    movel([0.074440, -1.320583, -2.610571, -0.781234, 1.570796, 1.645237],accel_mss,speed_ms,0,blend_radius_m)
    movel([0.074315, -1.320855, -2.610402, -0.781132, 1.570796, 1.645112],accel_mss,speed_ms,0,blend_radius_m)
    movel([0.073757, -1.321736, -2.609852, -0.780801, 1.570796, 1.644553],accel_mss,speed_ms,0,blend_radius_m)
    movel([0.073104, -1.322417, -2.609427, -0.780545, 1.570796, 1.643900],accel_mss,speed_ms,0,blend_radius_m)
    movel([0.072314, -1.322927, -2.609108, -0.780355, 1.570796, 1.643111],accel_mss,speed_ms,0,blend_radius_m)
    movel([0.071362, -1.323294, -2.608878, -0.780217, 1.570796, 1.642159],accel_mss,speed_ms,0,blend_radius_m)
    movel([0.070869, -1.323423, -2.608797, -0.780169, 1.570796, 1.641665],accel_mss,speed_ms,0,blend_radius_m)
    movel([0.070526, -1.323474, -2.608765, -0.780150, 1.570796, 1.641322],accel_mss,speed_ms,0,blend_radius_m)
    movel([0.070234, -1.323465, -2.608771, -0.780154, 1.570796, 1.641030],accel_mss,speed_ms,0,blend_radius_m)
    movel([0.069916, -1.323397, -2.608813, -0.780179, 1.570796, 1.640712],accel_mss,speed_ms,0,blend_radius_m)
    movel([0.069099, -1.322793, -2.609191, -0.780404, 1.570796, 1.639896],accel_mss,speed_ms,0,blend_radius_m)
    movel([0.068874, -1.321709, -2.609869, -0.780811, 1.570796, 1.639671],accel_mss,speed_ms,0,blend_radius_m)
    movel([0.069290, -1.320407, -2.610681, -0.781301, 1.570796, 1.640086],accel_mss,speed_ms,0,blend_radius_m)
    movel([0.070255, -1.319201, -2.611431, -0.781757, 1.570796, 1.641051],accel_mss,speed_ms,0,blend_radius_m)
    movel([0.070604, -1.318907, -2.611613, -0.781868, 1.570796, 1.641400],accel_mss,speed_ms,0,blend_radius_m)
    movel([0.070915, -1.318695, -2.611745, -0.781949, 1.570796, 1.641711],accel_mss,speed_ms,0,blend_radius_m)
    movel([0.071271, -1.318512, -2.611859, -0.782018, 1.570796, 1.642068],accel_mss,speed_ms,0,blend_radius_m)
    movel([0.071774, -1.318306, -2.611986, -0.782096, 1.570796, 1.642570],accel_mss,speed_ms,0,blend_radius_m)
    movel([0.072472, -1.318085, -2.612123, -0.782180, 1.570796, 1.643268],accel_mss,speed_ms,0,blend_radius_m)
    movel([0.073056, -1.318004, -2.612174, -0.782212, 1.570796, 1.643852],accel_mss,speed_ms,0,blend_radius_m)
    movel([0.073553, -1.318057, -2.612141, -0.782191, 1.570796, 1.644349],accel_mss,speed_ms,0,blend_radius_m)
    movel([0.073982, -1.318249, -2.612022, -0.782118, 1.570796, 1.644779],accel_mss,speed_ms,0,blend_radius_m)
    movel([0.074267, -1.318512, -2.611859, -0.782018, 1.570796, 1.645063],accel_mss,speed_ms,0,blend_radius_m)
    movel([0.074500, -1.318909, -2.611612, -0.781868, 1.570796, 1.645296],accel_mss,speed_ms,0,blend_radius_m)
    movel([0.074648, -1.319355, -2.611336, -0.781699, 1.570796, 1.645444],accel_mss,speed_ms,0,blend_radius_m)
    speed_ms = 0.003
    movel([0.074648, -1.322804, -2.612923, -0.776662, 1.570796, 1.645444],accel_mss,speed_ms,0,blend_radius_m)
    speed_ms = 0.007
    movel([0.074675, -1.323216, -2.612666, -0.776507, 1.570796, 1.645472],accel_mss,speed_ms,0,blend_radius_m)
    movel([0.074553, -1.323727, -2.612346, -0.776316, 1.570796, 1.645349],accel_mss,speed_ms,0,blend_radius_m)
    movel([0.074440, -1.324030, -2.612157, -0.776203, 1.570796, 1.645237],accel_mss,speed_ms,0,blend_radius_m)
    movel([0.074315, -1.324301, -2.611987, -0.776101, 1.570796, 1.645112],accel_mss,speed_ms,0,blend_radius_m)
    movel([0.073757, -1.325180, -2.611436, -0.775773, 1.570796, 1.644553],accel_mss,speed_ms,0,blend_radius_m)
    movel([0.073104, -1.325859, -2.611009, -0.775521, 1.570796, 1.643900],accel_mss,speed_ms,0,blend_radius_m)
    movel([0.072314, -1.326368, -2.610689, -0.775332, 1.570796, 1.643111],accel_mss,speed_ms,0,blend_radius_m)
    movel([0.071362, -1.326734, -2.610459, -0.775196, 1.570796, 1.642159],accel_mss,speed_ms,0,blend_radius_m)
    movel([0.070869, -1.326862, -2.610378, -0.775149, 1.570796, 1.641665],accel_mss,speed_ms,0,blend_radius_m)
    movel([0.070526, -1.326913, -2.610346, -0.775130, 1.570796, 1.641322],accel_mss,speed_ms,0,blend_radius_m)
    movel([0.070234, -1.326904, -2.610351, -0.775133, 1.570796, 1.641030],accel_mss,speed_ms,0,blend_radius_m)
    movel([0.069916, -1.326837, -2.610394, -0.775159, 1.570796, 1.640712],accel_mss,speed_ms,0,blend_radius_m)
    movel([0.069099, -1.326234, -2.610773, -0.775382, 1.570796, 1.639896],accel_mss,speed_ms,0,blend_radius_m)
    movel([0.068874, -1.325153, -2.611453, -0.775784, 1.570796, 1.639671],accel_mss,speed_ms,0,blend_radius_m)
    movel([0.069290, -1.323854, -2.612267, -0.776268, 1.570796, 1.640086],accel_mss,speed_ms,0,blend_radius_m)
    movel([0.070255, -1.322650, -2.613019, -0.776720, 1.570796, 1.641051],accel_mss,speed_ms,0,blend_radius_m)
    movel([0.070604, -1.322358, -2.613202, -0.776829, 1.570796, 1.641400],accel_mss,speed_ms,0,blend_radius_m)
    movel([0.070915, -1.322146, -2.613334, -0.776909, 1.570796, 1.641711],accel_mss,speed_ms,0,blend_radius_m)
    movel([0.071271, -1.321963, -2.613448, -0.776978, 1.570796, 1.642068],accel_mss,speed_ms,0,blend_radius_m)
    movel([0.071774, -1.321758, -2.613576, -0.777055, 1.570796, 1.642570],accel_mss,speed_ms,0,blend_radius_m)
    movel([0.072472, -1.321538, -2.613713, -0.777138, 1.570796, 1.643268],accel_mss,speed_ms,0,blend_radius_m)
    movel([0.073056, -1.321456, -2.613764, -0.777169, 1.570796, 1.643852],accel_mss,speed_ms,0,blend_radius_m)
    movel([0.073553, -1.321509, -2.613731, -0.777149, 1.570796, 1.644349],accel_mss,speed_ms,0,blend_radius_m)
    movel([0.073982, -1.321701, -2.613611, -0.777077, 1.570796, 1.644779],accel_mss,speed_ms,0,blend_radius_m)
    movel([0.074267, -1.321963, -2.613448, -0.776978, 1.570796, 1.645063],accel_mss,speed_ms,0,blend_radius_m)
    movel([0.074500, -1.322359, -2.613201, -0.776829, 1.570796, 1.645296],accel_mss,speed_ms,0,blend_radius_m)
    movel([0.074648, -1.322804, -2.612923, -0.776662, 1.570796, 1.645444],accel_mss,speed_ms,0,blend_radius_m)
    speed_ms = 0.003
    movel([0.074648, -1.309165, -2.606523, -0.796701, 1.570796, 1.645444],accel_mss,speed_ms,0,blend_radius_m)
    speed_ms = 1.000
    movel([0.074648, -1.283142, -2.593332, -0.835915, 1.570796, 1.645444],accel_mss,speed_ms,0,blend_radius_m)
    movel([0.075024, -1.282687, -2.593600, -0.836102, 1.570796, 1.645820],accel_mss,speed_ms,0,blend_radius_m)
    movel([0.075024, -1.308718, -2.606796, -0.796875, 1.570796, 1.645820],accel_mss,speed_ms,0,blend_radius_m)
    speed_ms = 0.003
    movel([0.075024, -1.318910, -2.611612, -0.781867, 1.570796, 1.645820],accel_mss,speed_ms,0,blend_radius_m)
    speed_ms = 0.007
    movel([0.075085, -1.319510, -2.611239, -0.781640, 1.570796, 1.645881],accel_mss,speed_ms,0,blend_radius_m)
    movel([0.074948, -1.320246, -2.610781, -0.781362, 1.570796, 1.645744],accel_mss,speed_ms,0,blend_radius_m)
    movel([0.074641, -1.321022, -2.610298, -0.781069, 1.570796, 1.645437],accel_mss,speed_ms,0,blend_radius_m)
    movel([0.074198, -1.321742, -2.609848, -0.780798, 1.570796, 1.644994],accel_mss,speed_ms,0,blend_radius_m)
    movel([0.073687, -1.322309, -2.609494, -0.780586, 1.570796, 1.644483],accel_mss,speed_ms,0,blend_radius_m)
    movel([0.073025, -1.322849, -2.609156, -0.780384, 1.570796, 1.643822],accel_mss,speed_ms,0,blend_radius_m)
    movel([0.072291, -1.323304, -2.608871, -0.780213, 1.570796, 1.643087],accel_mss,speed_ms,0,blend_radius_m)
    movel([0.071565, -1.323618, -2.608674, -0.780096, 1.570796, 1.642362],accel_mss,speed_ms,0,blend_radius_m)
    movel([0.070602, -1.323847, -2.608531, -0.780011, 1.570796, 1.641398],accel_mss,speed_ms,0,blend_radius_m)
    movel([0.069813, -1.323830, -2.608542, -0.780017, 1.570796, 1.640609],accel_mss,speed_ms,0,blend_radius_m)
    movel([0.069187, -1.323555, -2.608714, -0.780120, 1.570796, 1.639984],accel_mss,speed_ms,0,blend_radius_m)
    movel([0.068697, -1.323026, -2.609045, -0.780317, 1.570796, 1.639493],accel_mss,speed_ms,0,blend_radius_m)
    movel([0.068546, -1.322743, -2.609223, -0.780423, 1.570796, 1.639343],accel_mss,speed_ms,0,blend_radius_m)
    movel([0.068478, -1.322487, -2.609383, -0.780519, 1.570796, 1.639274],accel_mss,speed_ms,0,blend_radius_m)
    movel([0.068472, -1.322167, -2.609583, -0.780639, 1.570796, 1.639268],accel_mss,speed_ms,0,blend_radius_m)
    movel([0.068526, -1.321647, -2.609908, -0.780834, 1.570796, 1.639322],accel_mss,speed_ms,0,blend_radius_m)
    movel([0.068607, -1.321120, -2.610237, -0.781032, 1.570796, 1.639403],accel_mss,speed_ms,0,blend_radius_m)
    movel([0.068702, -1.320774, -2.610453, -0.781163, 1.570796, 1.639499],accel_mss,speed_ms,0,blend_radius_m)
    movel([0.068847, -1.320465, -2.610645, -0.781279, 1.570796, 1.639644],accel_mss,speed_ms,0,blend_radius_m)
    movel([0.069093, -1.320085, -2.610882, -0.781423, 1.570796, 1.639889],accel_mss,speed_ms,0,blend_radius_m)
    movel([0.069307, -1.319800, -2.611058, -0.781530, 1.570796, 1.640103],accel_mss,speed_ms,0,blend_radius_m)
    movel([0.069588, -1.319471, -2.611263, -0.781655, 1.570796, 1.640384],accel_mss,speed_ms,0,blend_radius_m)
    movel([0.069884, -1.319150, -2.611463, -0.781776, 1.570796, 1.640680],accel_mss,speed_ms,0,blend_radius_m)
    movel([0.070148, -1.318894, -2.611621, -0.781873, 1.570796, 1.640945],accel_mss,speed_ms,0,blend_radius_m)
    movel([0.070517, -1.318583, -2.611815, -0.781991, 1.570796, 1.641314],accel_mss,speed_ms,0,blend_radius_m)
    movel([0.070837, -1.318370, -2.611946, -0.782072, 1.570796, 1.641633],accel_mss,speed_ms,0,blend_radius_m)
    movel([0.071214, -1.318184, -2.612062, -0.782143, 1.570796, 1.642011],accel_mss,speed_ms,0,blend_radius_m)
    movel([0.071809, -1.317950, -2.612207, -0.782232, 1.570796, 1.642605],accel_mss,speed_ms,0,blend_radius_m)
    movel([0.072379, -1.317746, -2.612333, -0.782309, 1.570796, 1.643176],accel_mss,speed_ms,0,blend_radius_m)
    movel([0.072764, -1.317643, -2.612397, -0.782349, 1.570796, 1.643560],accel_mss,speed_ms,0,blend_radius_m)
    movel([0.073074, -1.317602, -2.612422, -0.782364, 1.570796, 1.643870],accel_mss,speed_ms,0,blend_radius_m)
    movel([0.073396, -1.317616, -2.612414, -0.782359, 1.570796, 1.644192],accel_mss,speed_ms,0,blend_radius_m)
    movel([0.073967, -1.317754, -2.612329, -0.782307, 1.570796, 1.644763],accel_mss,speed_ms,0,blend_radius_m)
    movel([0.074437, -1.318021, -2.612163, -0.782205, 1.570796, 1.645234],accel_mss,speed_ms,0,blend_radius_m)
    movel([0.074794, -1.318414, -2.611920, -0.782056, 1.570796, 1.645591],accel_mss,speed_ms,0,blend_radius_m)
    movel([0.075024, -1.318910, -2.611612, -0.781867, 1.570796, 1.645820],accel_mss,speed_ms,0,blend_radius_m)
    speed_ms = 0.003
    movel([0.075024, -1.322360, -2.613200, -0.776828, 1.570796, 1.645820],accel_mss,speed_ms,0,blend_radius_m)
    speed_ms = 0.007
    movel([0.075085, -1.322959, -2.612826, -0.776604, 1.570796, 1.645881],accel_mss,speed_ms,0,blend_radius_m)
    movel([0.074948, -1.323693, -2.612367, -0.776328, 1.570796, 1.645744],accel_mss,speed_ms,0,blend_radius_m)
    movel([0.074641, -1.324467, -2.611883, -0.776039, 1.570796, 1.645437],accel_mss,speed_ms,0,blend_radius_m)
    movel([0.074198, -1.325186, -2.611432, -0.775771, 1.570796, 1.644994],accel_mss,speed_ms,0,blend_radius_m)
    movel([0.073687, -1.325751, -2.611077, -0.775561, 1.570796, 1.644483],accel_mss,speed_ms,0,blend_radius_m)
    movel([0.073025, -1.326290, -2.610738, -0.775361, 1.570796, 1.643822],accel_mss,speed_ms,0,blend_radius_m)
    movel([0.072291, -1.326744, -2.610452, -0.775193, 1.570796, 1.643087],accel_mss,speed_ms,0,blend_radius_m)
    movel([0.071565, -1.327058, -2.610255, -0.775077, 1.570796, 1.642362],accel_mss,speed_ms,0,blend_radius_m)
    movel([0.070602, -1.327285, -2.610111, -0.774992, 1.570796, 1.641398],accel_mss,speed_ms,0,blend_radius_m)
    movel([0.069813, -1.327269, -2.610122, -0.774999, 1.570796, 1.640609],accel_mss,speed_ms,0,blend_radius_m)
    movel([0.069187, -1.326994, -2.610295, -0.775100, 1.570796, 1.639984],accel_mss,speed_ms,0,blend_radius_m)
    movel([0.068697, -1.326467, -2.610627, -0.775296, 1.570796, 1.639493],accel_mss,speed_ms,0,blend_radius_m)
    movel([0.068546, -1.326184, -2.610804, -0.775400, 1.570796, 1.639343],accel_mss,speed_ms,0,blend_radius_m)
    movel([0.068478, -1.325929, -2.610965, -0.775495, 1.570796, 1.639274],accel_mss,speed_ms,0,blend_radius_m)
    movel([0.068472, -1.325610, -2.611166, -0.775614, 1.570796, 1.639268],accel_mss,speed_ms,0,blend_radius_m)
    movel([0.068526, -1.325091, -2.611492, -0.775807, 1.570796, 1.639322],accel_mss,speed_ms,0,blend_radius_m)
    movel([0.068607, -1.324565, -2.611821, -0.776003, 1.570796, 1.639403],accel_mss,speed_ms,0,blend_radius_m)
    movel([0.068702, -1.324220, -2.612038, -0.776132, 1.570796, 1.639499],accel_mss,speed_ms,0,blend_radius_m)
    movel([0.068847, -1.323912, -2.612230, -0.776247, 1.570796, 1.639644],accel_mss,speed_ms,0,blend_radius_m)
    movel([0.069093, -1.323532, -2.612468, -0.776389, 1.570796, 1.639889],accel_mss,speed_ms,0,blend_radius_m)
    movel([0.069307, -1.323249, -2.612645, -0.776495, 1.570796, 1.640103],accel_mss,speed_ms,0,blend_radius_m)
    movel([0.069588, -1.322920, -2.612851, -0.776618, 1.570796, 1.640384],accel_mss,speed_ms,0,blend_radius_m)
    movel([0.069884, -1.322600, -2.613051, -0.776738, 1.570796, 1.640680],accel_mss,speed_ms,0,blend_radius_m)
    movel([0.070148, -1.322345, -2.613210, -0.776834, 1.570796, 1.640945],accel_mss,speed_ms,0,blend_radius_m)
    movel([0.070517, -1.322034, -2.613404, -0.776951, 1.570796, 1.641314],accel_mss,speed_ms,0,blend_radius_m)
    movel([0.070837, -1.321822, -2.613536, -0.777031, 1.570796, 1.641633],accel_mss,speed_ms,0,blend_radius_m)
    movel([0.071214, -1.321636, -2.613652, -0.777101, 1.570796, 1.642011],accel_mss,speed_ms,0,blend_radius_m)
    movel([0.071809, -1.321402, -2.613797, -0.777189, 1.570796, 1.642605],accel_mss,speed_ms,0,blend_radius_m)
    movel([0.072379, -1.321200, -2.613923, -0.777266, 1.570796, 1.643176],accel_mss,speed_ms,0,blend_radius_m)
    movel([0.072764, -1.321096, -2.613988, -0.777305, 1.570796, 1.643560],accel_mss,speed_ms,0,blend_radius_m)
    movel([0.073074, -1.321056, -2.614013, -0.777320, 1.570796, 1.643870],accel_mss,speed_ms,0,blend_radius_m)
    movel([0.073396, -1.321069, -2.614005, -0.777315, 1.570796, 1.644192],accel_mss,speed_ms,0,blend_radius_m)
    movel([0.073967, -1.321207, -2.613919, -0.777263, 1.570796, 1.644763],accel_mss,speed_ms,0,blend_radius_m)
    movel([0.074437, -1.321474, -2.613753, -0.777162, 1.570796, 1.645234],accel_mss,speed_ms,0,blend_radius_m)
    movel([0.074794, -1.321865, -2.613509, -0.777015, 1.570796, 1.645591],accel_mss,speed_ms,0,blend_radius_m)
    movel([0.075024, -1.322360, -2.613200, -0.776828, 1.570796, 1.645820],accel_mss,speed_ms,0,blend_radius_m)
    speed_ms = 0.003
    movel([0.075024, -1.308718, -2.606796, -0.796875, 1.570796, 1.645820],accel_mss,speed_ms,0,blend_radius_m)
    speed_ms = 1.000
    movel([0.075024, -1.282687, -2.593600, -0.836102, 1.570796, 1.645820],accel_mss,speed_ms,0,blend_radius_m)
    movel([0.074027, -1.283141, -2.593332, -0.835916, 1.570796, 1.644824],accel_mss,speed_ms,0,blend_radius_m)
    movel([0.074027, -1.309165, -2.606523, -0.796701, 1.570796, 1.644824],accel_mss,speed_ms,0,blend_radius_m)
    speed_ms = 0.003
    movel([0.074027, -1.319354, -2.611336, -0.781699, 1.570796, 1.644824],accel_mss,speed_ms,0,blend_radius_m)
    speed_ms = 0.007
    movel([0.073556, -1.319849, -2.611028, -0.781512, 1.570796, 1.644352],accel_mss,speed_ms,0,blend_radius_m)
    movel([0.072865, -1.320341, -2.610722, -0.781326, 1.570796, 1.643661],accel_mss,speed_ms,0,blend_radius_m)
    movel([0.072601, -1.320557, -2.610588, -0.781244, 1.570796, 1.643397],accel_mss,speed_ms,0,blend_radius_m)
    movel([0.072444, -1.321001, -2.610311, -0.781077, 1.570796, 1.643240],accel_mss,speed_ms,0,blend_radius_m)
    movel([0.072443, -1.321758, -2.609838, -0.780792, 1.570796, 1.643239],accel_mss,speed_ms,0,blend_radius_m)
    movel([0.072434, -1.321990, -2.609693, -0.780705, 1.570796, 1.643230],accel_mss,speed_ms,0,blend_radius_m)
    movel([0.072327, -1.322242, -2.609536, -0.780611, 1.570796, 1.643123],accel_mss,speed_ms,0,blend_radius_m)
    movel([0.071996, -1.322298, -2.609501, -0.780590, 1.570796, 1.642792],accel_mss,speed_ms,0,blend_radius_m)
    movel([0.071795, -1.321918, -2.609739, -0.780733, 1.570796, 1.642591],accel_mss,speed_ms,0,blend_radius_m)
    movel([0.071704, -1.321719, -2.609863, -0.780807, 1.570796, 1.642500],accel_mss,speed_ms,0,blend_radius_m)
    movel([0.071601, -1.321544, -2.609972, -0.780873, 1.570796, 1.642397],accel_mss,speed_ms,0,blend_radius_m)
    movel([0.071406, -1.321373, -2.610079, -0.780937, 1.570796, 1.642202],accel_mss,speed_ms,0,blend_radius_m)
    movel([0.071079, -1.321469, -2.610019, -0.780901, 1.570796, 1.641875],accel_mss,speed_ms,0,blend_radius_m)
    movel([0.070562, -1.321740, -2.609850, -0.780799, 1.570796, 1.641358],accel_mss,speed_ms,0,blend_radius_m)
    movel([0.070211, -1.321941, -2.609724, -0.780724, 1.570796, 1.641007],accel_mss,speed_ms,0,blend_radius_m)
    movel([0.069848, -1.322070, -2.609644, -0.780675, 1.570796, 1.640644],accel_mss,speed_ms,0,blend_radius_m)
    movel([0.069610, -1.321995, -2.609690, -0.780703, 1.570796, 1.640407],accel_mss,speed_ms,0,blend_radius_m)
    movel([0.069744, -1.321703, -2.609873, -0.780813, 1.570796, 1.640540],accel_mss,speed_ms,0,blend_radius_m)
    movel([0.070057, -1.321421, -2.610049, -0.780919, 1.570796, 1.640853],accel_mss,speed_ms,0,blend_radius_m)
    movel([0.070500, -1.321122, -2.610236, -0.781032, 1.570796, 1.641296],accel_mss,speed_ms,0,blend_radius_m)
    movel([0.070910, -1.320839, -2.610412, -0.781138, 1.570796, 1.641707],accel_mss,speed_ms,0,blend_radius_m)
    movel([0.071115, -1.320581, -2.610573, -0.781235, 1.570796, 1.641911],accel_mss,speed_ms,0,blend_radius_m)
    movel([0.071162, -1.320290, -2.610754, -0.781345, 1.570796, 1.641958],accel_mss,speed_ms,0,blend_radius_m)
    movel([0.071051, -1.319883, -2.611007, -0.781499, 1.570796, 1.641848],accel_mss,speed_ms,0,blend_radius_m)
    movel([0.070960, -1.319617, -2.611172, -0.781599, 1.570796, 1.641757],accel_mss,speed_ms,0,blend_radius_m)
    movel([0.070970, -1.319306, -2.611366, -0.781717, 1.570796, 1.641766],accel_mss,speed_ms,0,blend_radius_m)
    movel([0.071177, -1.319020, -2.611543, -0.781825, 1.570796, 1.641973],accel_mss,speed_ms,0,blend_radius_m)
    movel([0.071466, -1.319017, -2.611546, -0.781827, 1.570796, 1.642262],accel_mss,speed_ms,0,blend_radius_m)
    movel([0.071655, -1.319206, -2.611428, -0.781755, 1.570796, 1.642451],accel_mss,speed_ms,0,blend_radius_m)
    movel([0.071802, -1.319519, -2.611233, -0.781636, 1.570796, 1.642598],accel_mss,speed_ms,0,blend_radius_m)
    movel([0.071941, -1.319865, -2.611019, -0.781506, 1.570796, 1.642737],accel_mss,speed_ms,0,blend_radius_m)
    movel([0.072115, -1.319984, -2.610944, -0.781461, 1.570796, 1.642911],accel_mss,speed_ms,0,blend_radius_m)
    movel([0.072792, -1.319712, -2.611113, -0.781564, 1.570796, 1.643588],accel_mss,speed_ms,0,blend_radius_m)
    movel([0.073214, -1.319464, -2.611268, -0.781657, 1.570796, 1.644010],accel_mss,speed_ms,0,blend_radius_m)
    movel([0.073566, -1.319296, -2.611372, -0.781721, 1.570796, 1.644362],accel_mss,speed_ms,0,blend_radius_m)
    movel([0.073838, -1.319207, -2.611427, -0.781754, 1.570796, 1.644634],accel_mss,speed_ms,0,blend_radius_m)
    movel([0.074027, -1.319354, -2.611336, -0.781699, 1.570796, 1.644824],accel_mss,speed_ms,0,blend_radius_m)
    speed_ms = 0.003
    movel([0.074027, -1.322803, -2.612924, -0.776662, 1.570796, 1.644824],accel_mss,speed_ms,0,blend_radius_m)
    speed_ms = 0.007
    movel([0.073556, -1.323297, -2.612615, -0.776477, 1.570796, 1.644352],accel_mss,speed_ms,0,blend_radius_m)
    movel([0.072865, -1.323788, -2.612308, -0.776293, 1.570796, 1.643661],accel_mss,speed_ms,0,blend_radius_m)
    movel([0.072601, -1.324003, -2.612173, -0.776212, 1.570796, 1.643397],accel_mss,speed_ms,0,blend_radius_m)
    movel([0.072444, -1.324446, -2.611896, -0.776047, 1.570796, 1.643240],accel_mss,speed_ms,0,blend_radius_m)
    movel([0.072443, -1.325202, -2.611422, -0.775765, 1.570796, 1.643239],accel_mss,speed_ms,0,blend_radius_m)
    movel([0.072434, -1.325433, -2.611276, -0.775679, 1.570796, 1.643230],accel_mss,speed_ms,0,blend_radius_m)
    movel([0.072327, -1.325684, -2.611119, -0.775586, 1.570796, 1.643123],accel_mss,speed_ms,0,blend_radius_m)
    movel([0.071996, -1.325740, -2.611084, -0.775565, 1.570796, 1.642792],accel_mss,speed_ms,0,blend_radius_m)
    movel([0.071795, -1.325361, -2.611322, -0.775706, 1.570796, 1.642591],accel_mss,speed_ms,0,blend_radius_m)
    movel([0.071704, -1.325162, -2.611447, -0.775780, 1.570796, 1.642500],accel_mss,speed_ms,0,blend_radius_m)
    movel([0.071601, -1.324988, -2.611556, -0.775845, 1.570796, 1.642397],accel_mss,speed_ms,0,blend_radius_m)
    movel([0.071406, -1.324817, -2.611663, -0.775908, 1.570796, 1.642202],accel_mss,speed_ms,0,blend_radius_m)
    movel([0.071079, -1.324913, -2.611603, -0.775873, 1.570796, 1.641875],accel_mss,speed_ms,0,blend_radius_m)
    movel([0.070562, -1.325183, -2.611434, -0.775772, 1.570796, 1.641358],accel_mss,speed_ms,0,blend_radius_m)
    movel([0.070211, -1.325384, -2.611307, -0.775697, 1.570796, 1.641007],accel_mss,speed_ms,0,blend_radius_m)
    movel([0.069848, -1.325513, -2.611227, -0.775650, 1.570796, 1.640644],accel_mss,speed_ms,0,blend_radius_m)
    movel([0.069610, -1.325438, -2.611273, -0.775677, 1.570796, 1.640407],accel_mss,speed_ms,0,blend_radius_m)
    movel([0.069744, -1.325147, -2.611456, -0.775786, 1.570796, 1.640540],accel_mss,speed_ms,0,blend_radius_m)
    movel([0.070057, -1.324865, -2.611633, -0.775891, 1.570796, 1.640853],accel_mss,speed_ms,0,blend_radius_m)
    movel([0.070500, -1.324567, -2.611820, -0.776002, 1.570796, 1.641296],accel_mss,speed_ms,0,blend_radius_m)
    movel([0.070910, -1.324284, -2.611997, -0.776107, 1.570796, 1.641707],accel_mss,speed_ms,0,blend_radius_m)
    movel([0.071115, -1.324028, -2.612158, -0.776203, 1.570796, 1.641911],accel_mss,speed_ms,0,blend_radius_m)
    movel([0.071162, -1.323737, -2.612340, -0.776312, 1.570796, 1.641958],accel_mss,speed_ms,0,blend_radius_m)
    movel([0.071051, -1.323331, -2.612594, -0.776464, 1.570796, 1.641848],accel_mss,speed_ms,0,blend_radius_m)
    movel([0.070960, -1.323066, -2.612759, -0.776563, 1.570796, 1.641757],accel_mss,speed_ms,0,blend_radius_m)
    movel([0.070970, -1.322756, -2.612953, -0.776680, 1.570796, 1.641766],accel_mss,speed_ms,0,blend_radius_m)
    movel([0.071177, -1.322470, -2.613132, -0.776787, 1.570796, 1.641973],accel_mss,speed_ms,0,blend_radius_m)
    movel([0.071466, -1.322467, -2.613134, -0.776789, 1.570796, 1.642262],accel_mss,speed_ms,0,blend_radius_m)
    movel([0.071655, -1.322656, -2.613016, -0.776717, 1.570796, 1.642451],accel_mss,speed_ms,0,blend_radius_m)
    movel([0.071802, -1.322968, -2.612821, -0.776600, 1.570796, 1.642598],accel_mss,speed_ms,0,blend_radius_m)
    movel([0.071941, -1.323313, -2.612605, -0.776471, 1.570796, 1.642737],accel_mss,speed_ms,0,blend_radius_m)
    movel([0.072115, -1.323432, -2.612531, -0.776426, 1.570796, 1.642911],accel_mss,speed_ms,0,blend_radius_m)
    movel([0.072792, -1.323160, -2.612701, -0.776528, 1.570796, 1.643588],accel_mss,speed_ms,0,blend_radius_m)
    movel([0.073214, -1.322913, -2.612855, -0.776621, 1.570796, 1.644010],accel_mss,speed_ms,0,blend_radius_m)
    movel([0.073566, -1.322746, -2.612960, -0.776684, 1.570796, 1.644362],accel_mss,speed_ms,0,blend_radius_m)
    movel([0.073838, -1.322657, -2.613015, -0.776717, 1.570796, 1.644634],accel_mss,speed_ms,0,blend_radius_m)
    movel([0.074027, -1.322803, -2.612924, -0.776662, 1.570796, 1.644824],accel_mss,speed_ms,0,blend_radius_m)
    speed_ms = 0.003
    movel([0.074027, -1.309165, -2.606523, -0.796701, 1.570796, 1.644824],accel_mss,speed_ms,0,blend_radius_m)
    speed_ms = 1.000
    movel([0.074027, -1.283141, -2.593332, -0.835916, 1.570796, 1.644824],accel_mss,speed_ms,0,blend_radius_m)
    movel([0.071023, -1.278128, -2.596274, -0.837987, 1.570796, 1.641819],accel_mss,speed_ms,0,blend_radius_m)
    movel([0.071023, -1.304226, -2.609531, -0.798633, 1.570796, 1.641819],accel_mss,speed_ms,0,blend_radius_m)
    speed_ms = 0.003
    movel([0.071023, -1.314448, -2.614368, -0.783573, 1.570796, 1.641819],accel_mss,speed_ms,0,blend_radius_m)
    speed_ms = 0.007
    movel([0.069147, -1.315811, -2.613529, -0.783049, 1.570796, 1.639943],accel_mss,speed_ms,0,blend_radius_m)
    movel([0.068357, -1.316304, -2.613225, -0.782860, 1.570796, 1.639153],accel_mss,speed_ms,0,blend_radius_m)
    movel([0.067918, -1.316419, -2.613154, -0.782816, 1.570796, 1.638715],accel_mss,speed_ms,0,blend_radius_m)
    movel([0.067617, -1.316265, -2.613249, -0.782875, 1.570796, 1.638413],accel_mss,speed_ms,0,blend_radius_m)
    movel([0.067573, -1.316019, -2.613400, -0.782969, 1.570796, 1.638369],accel_mss,speed_ms,0,blend_radius_m)
    movel([0.067713, -1.315740, -2.613573, -0.783076, 1.570796, 1.638510],accel_mss,speed_ms,0,blend_radius_m)
    movel([0.068093, -1.315373, -2.613799, -0.783217, 1.570796, 1.638889],accel_mss,speed_ms,0,blend_radius_m)
    movel([0.068839, -1.314811, -2.614145, -0.783433, 1.570796, 1.639635],accel_mss,speed_ms,0,blend_radius_m)
    movel([0.070239, -1.313837, -2.614744, -0.783808, 1.570796, 1.641035],accel_mss,speed_ms,0,blend_radius_m)
    movel([0.070997, -1.313439, -2.614988, -0.783962, 1.570796, 1.641793],accel_mss,speed_ms,0,blend_radius_m)
    movel([0.071373, -1.313456, -2.614977, -0.783955, 1.570796, 1.642169],accel_mss,speed_ms,0,blend_radius_m)
    movel([0.071504, -1.313791, -2.614772, -0.783826, 1.570796, 1.642300],accel_mss,speed_ms,0,blend_radius_m)
    movel([0.071385, -1.314116, -2.614572, -0.783701, 1.570796, 1.642181],accel_mss,speed_ms,0,blend_radius_m)
    movel([0.071023, -1.314448, -2.614368, -0.783573, 1.570796, 1.641819],accel_mss,speed_ms,0,blend_radius_m)
    speed_ms = 0.003
    movel([0.071023, -1.317909, -2.615964, -0.778516, 1.570796, 1.641819],accel_mss,speed_ms,0,blend_radius_m)
    speed_ms = 0.007
    movel([0.069147, -1.319269, -2.615122, -0.777998, 1.570796, 1.639943],accel_mss,speed_ms,0,blend_radius_m)
    movel([0.068357, -1.319761, -2.614817, -0.777811, 1.570796, 1.639153],accel_mss,speed_ms,0,blend_radius_m)
    movel([0.067918, -1.319875, -2.614746, -0.777767, 1.570796, 1.638715],accel_mss,speed_ms,0,blend_radius_m)
    movel([0.067617, -1.319722, -2.614841, -0.777825, 1.570796, 1.638413],accel_mss,speed_ms,0,blend_radius_m)
    movel([0.067573, -1.319477, -2.614994, -0.777919, 1.570796, 1.638369],accel_mss,speed_ms,0,blend_radius_m)
    movel([0.067713, -1.319198, -2.615166, -0.778024, 1.570796, 1.638510],accel_mss,speed_ms,0,blend_radius_m)
    movel([0.068093, -1.318831, -2.615394, -0.778164, 1.570796, 1.638889],accel_mss,speed_ms,0,blend_radius_m)
    movel([0.068839, -1.318271, -2.615740, -0.778378, 1.570796, 1.639635],accel_mss,speed_ms,0,blend_radius_m)
    movel([0.070239, -1.317299, -2.616341, -0.778749, 1.570796, 1.641035],accel_mss,speed_ms,0,blend_radius_m)
    movel([0.070997, -1.316902, -2.616586, -0.778901, 1.570796, 1.641793],accel_mss,speed_ms,0,blend_radius_m)
    movel([0.071373, -1.316919, -2.616575, -0.778895, 1.570796, 1.642169],accel_mss,speed_ms,0,blend_radius_m)
    movel([0.071504, -1.317253, -2.616369, -0.778767, 1.570796, 1.642300],accel_mss,speed_ms,0,blend_radius_m)
    movel([0.071385, -1.317578, -2.616169, -0.778642, 1.570796, 1.642181],accel_mss,speed_ms,0,blend_radius_m)
    movel([0.071023, -1.317909, -2.615964, -0.778516, 1.570796, 1.641819],accel_mss,speed_ms,0,blend_radius_m)
    speed_ms = 0.003
    movel([0.071023, -1.304226, -2.609531, -0.798633, 1.570796, 1.641819],accel_mss,speed_ms,0,blend_radius_m)
    speed_ms = 1.000
    movel([0.071023, -1.278128, -2.596274, -0.837987, 1.570796, 1.641819],accel_mss,speed_ms,0,blend_radius_m)
    movel([0.070234, -1.277001, -2.596932, -0.838457, 1.570796, 1.641030],accel_mss,speed_ms,0,blend_radius_m)
    movel([0.070234, -1.303115, -2.610203, -0.799072, 1.570796, 1.641030],accel_mss,speed_ms,0,blend_radius_m)
    speed_ms = 0.003
    movel([0.070234, -1.313344, -2.615046, -0.783999, 1.570796, 1.641030],accel_mss,speed_ms,0,blend_radius_m)
    speed_ms = 0.007
    movel([0.069690, -1.313736, -2.614806, -0.783847, 1.570796, 1.640486],accel_mss,speed_ms,0,blend_radius_m)
    movel([0.069350, -1.313960, -2.614668, -0.783761, 1.570796, 1.640146],accel_mss,speed_ms,0,blend_radius_m)
    movel([0.068982, -1.314205, -2.614518, -0.783667, 1.570796, 1.639778],accel_mss,speed_ms,0,blend_radius_m)
    movel([0.068608, -1.314463, -2.614359, -0.783567, 1.570796, 1.639404],accel_mss,speed_ms,0,blend_radius_m)
    movel([0.068272, -1.314701, -2.614212, -0.783475, 1.570796, 1.639068],accel_mss,speed_ms,0,blend_radius_m)
    movel([0.067748, -1.315091, -2.613973, -0.783325, 1.570796, 1.638544],accel_mss,speed_ms,0,blend_radius_m)
    movel([0.067368, -1.315127, -2.613951, -0.783312, 1.570796, 1.638164],accel_mss,speed_ms,0,blend_radius_m)
    movel([0.067208, -1.314950, -2.614059, -0.783379, 1.570796, 1.638004],accel_mss,speed_ms,0,blend_radius_m)
    movel([0.067125, -1.314520, -2.614324, -0.783545, 1.570796, 1.637921],accel_mss,speed_ms,0,blend_radius_m)
    movel([0.067331, -1.314004, -2.614641, -0.783744, 1.570796, 1.638127],accel_mss,speed_ms,0,blend_radius_m)
    movel([0.067860, -1.313393, -2.615016, -0.783980, 1.570796, 1.638656],accel_mss,speed_ms,0,blend_radius_m)
    movel([0.068714, -1.312682, -2.615452, -0.784255, 1.570796, 1.639510],accel_mss,speed_ms,0,blend_radius_m)
    movel([0.069595, -1.312087, -2.615816, -0.784486, 1.570796, 1.640391],accel_mss,speed_ms,0,blend_radius_m)
    movel([0.070212, -1.311846, -2.615963, -0.784579, 1.570796, 1.641008],accel_mss,speed_ms,0,blend_radius_m)
    movel([0.070613, -1.311926, -2.615915, -0.784548, 1.570796, 1.641409],accel_mss,speed_ms,0,blend_radius_m)
    movel([0.070831, -1.312303, -2.615684, -0.784402, 1.570796, 1.641627],accel_mss,speed_ms,0,blend_radius_m)
    movel([0.070900, -1.312683, -2.615452, -0.784255, 1.570796, 1.641697],accel_mss,speed_ms,0,blend_radius_m)
    movel([0.070811, -1.312966, -2.615278, -0.784145, 1.570796, 1.641607],accel_mss,speed_ms,0,blend_radius_m)
    movel([0.070439, -1.313152, -2.615164, -0.784073, 1.570796, 1.641236],accel_mss,speed_ms,0,blend_radius_m)
    speed_ms = 0.003
    movel([0.070234, -1.316808, -2.616644, -0.778937, 1.570796, 1.641030],accel_mss,speed_ms,0,blend_radius_m)
    speed_ms = 0.007
    movel([0.069690, -1.317199, -2.616403, -0.778788, 1.570796, 1.640486],accel_mss,speed_ms,0,blend_radius_m)
    movel([0.069350, -1.317422, -2.616265, -0.778702, 1.570796, 1.640146],accel_mss,speed_ms,0,blend_radius_m)
    movel([0.068982, -1.317666, -2.616114, -0.778609, 1.570796, 1.639778],accel_mss,speed_ms,0,blend_radius_m)
    movel([0.068608, -1.317924, -2.615955, -0.778510, 1.570796, 1.639404],accel_mss,speed_ms,0,blend_radius_m)
    movel([0.068272, -1.318162, -2.615808, -0.778419, 1.570796, 1.639068],accel_mss,speed_ms,0,blend_radius_m)
    movel([0.067748, -1.318551, -2.615567, -0.778271, 1.570796, 1.638544],accel_mss,speed_ms,0,blend_radius_m)
    movel([0.067368, -1.318586, -2.615545, -0.778257, 1.570796, 1.638164],accel_mss,speed_ms,0,blend_radius_m)
    movel([0.067208, -1.318410, -2.615654, -0.778325, 1.570796, 1.638004],accel_mss,speed_ms,0,blend_radius_m)
    movel([0.067125, -1.317980, -2.615920, -0.778489, 1.570796, 1.637921],accel_mss,speed_ms,0,blend_radius_m)
    movel([0.067331, -1.317466, -2.616238, -0.778685, 1.570796, 1.638127],accel_mss,speed_ms,0,blend_radius_m)
    movel([0.067860, -1.316857, -2.616614, -0.778919, 1.570796, 1.638656],accel_mss,speed_ms,0,blend_radius_m)
    movel([0.068714, -1.316147, -2.617051, -0.779191, 1.570796, 1.639510],accel_mss,speed_ms,0,blend_radius_m)
    movel([0.069595, -1.315553, -2.617416, -0.779420, 1.570796, 1.640391],accel_mss,speed_ms,0,blend_radius_m)
    movel([0.070212, -1.315313, -2.617564, -0.779512, 1.570796, 1.641008],accel_mss,speed_ms,0,blend_radius_m)
    movel([0.070613, -1.315393, -2.617515, -0.779481, 1.570796, 1.641409],accel_mss,speed_ms,0,blend_radius_m)
    movel([0.070831, -1.315769, -2.617283, -0.779336, 1.570796, 1.641627],accel_mss,speed_ms,0,blend_radius_m)
    movel([0.070900, -1.316148, -2.617050, -0.779191, 1.570796, 1.641697],accel_mss,speed_ms,0,blend_radius_m)
    movel([0.070811, -1.316431, -2.616876, -0.779082, 1.570796, 1.641607],accel_mss,speed_ms,0,blend_radius_m)
    movel([0.070439, -1.316616, -2.616762, -0.779011, 1.570796, 1.641236],accel_mss,speed_ms,0,blend_radius_m)
    speed_ms = 0.003
    movel([0.070234, -1.303115, -2.610203, -0.799072, 1.570796, 1.641030],accel_mss,speed_ms,0,blend_radius_m)
    speed_ms = 1.000
    movel([0.070234, -1.277001, -2.596932, -0.838457, 1.570796, 1.641030],accel_mss,speed_ms,0,blend_radius_m)
    movel([0.073982, -1.263429, -2.604724, -0.844235, 1.570796, 1.644779],accel_mss,speed_ms,0,blend_radius_m)
    movel([0.073982, -1.289735, -2.618173, -0.804481, 1.570796, 1.644779],accel_mss,speed_ms,0,blend_radius_m)
    speed_ms = 0.003
    movel([0.073982, -1.300051, -2.623084, -0.789254, 1.570796, 1.644779],accel_mss,speed_ms,0,blend_radius_m)
    speed_ms = 0.007
    movel([0.073932, -1.299789, -2.623240, -0.789360, 1.570796, 1.644728],accel_mss,speed_ms,0,blend_radius_m)
    movel([0.074261, -1.299549, -2.623383, -0.789457, 1.570796, 1.645057],accel_mss,speed_ms,0,blend_radius_m)
    movel([0.074673, -1.299325, -2.623517, -0.789548, 1.570796, 1.645470],accel_mss,speed_ms,0,blend_radius_m)
    movel([0.074331, -1.299356, -2.623498, -0.789535, 1.570796, 1.645127],accel_mss,speed_ms,0,blend_radius_m)
    movel([0.073782, -1.299594, -2.623356, -0.789439, 1.570796, 1.644579],accel_mss,speed_ms,0,blend_radius_m)
    movel([0.072985, -1.299872, -2.623191, -0.789326, 1.570796, 1.643781],accel_mss,speed_ms,0,blend_radius_m)
    movel([0.072179, -1.300125, -2.623040, -0.789224, 1.570796, 1.642975],accel_mss,speed_ms,0,blend_radius_m)
    movel([0.071902, -1.300103, -2.623053, -0.789233, 1.570796, 1.642698],accel_mss,speed_ms,0,blend_radius_m)
    movel([0.071682, -1.300397, -2.622877, -0.789114, 1.570796, 1.642478],accel_mss,speed_ms,0,blend_radius_m)
    movel([0.071302, -1.300592, -2.622761, -0.789035, 1.570796, 1.642098],accel_mss,speed_ms,0,blend_radius_m)
    movel([0.071480, -1.300308, -2.622931, -0.789150, 1.570796, 1.642277],accel_mss,speed_ms,0,blend_radius_m)
    movel([0.071194, -1.300365, -2.622897, -0.789127, 1.570796, 1.641991],accel_mss,speed_ms,0,blend_radius_m)
    movel([0.070917, -1.300543, -2.622791, -0.789055, 1.570796, 1.641714],accel_mss,speed_ms,0,blend_radius_m)
    movel([0.070724, -1.300383, -2.622886, -0.789120, 1.570796, 1.641520],accel_mss,speed_ms,0,blend_radius_m)
    movel([0.070555, -1.300212, -2.622988, -0.789189, 1.570796, 1.641352],accel_mss,speed_ms,0,blend_radius_m)
    movel([0.070266, -1.300204, -2.622993, -0.789192, 1.570796, 1.641063],accel_mss,speed_ms,0,blend_radius_m)
    movel([0.070498, -1.300295, -2.622938, -0.789155, 1.570796, 1.641294],accel_mss,speed_ms,0,blend_radius_m)
    movel([0.070207, -1.300506, -2.622813, -0.789070, 1.570796, 1.641004],accel_mss,speed_ms,0,blend_radius_m)
    movel([0.069999, -1.300433, -2.622856, -0.789100, 1.570796, 1.640795],accel_mss,speed_ms,0,blend_radius_m)
    movel([0.069864, -1.300276, -2.622950, -0.789163, 1.570796, 1.640660],accel_mss,speed_ms,0,blend_radius_m)
    movel([0.069616, -1.300492, -2.622821, -0.789076, 1.570796, 1.640412],accel_mss,speed_ms,0,blend_radius_m)
    movel([0.069394, -1.300421, -2.622863, -0.789105, 1.570796, 1.640190],accel_mss,speed_ms,0,blend_radius_m)
    movel([0.069164, -1.300073, -2.623071, -0.789245, 1.570796, 1.639960],accel_mss,speed_ms,0,blend_radius_m)
    movel([0.068809, -1.300112, -2.623048, -0.789229, 1.570796, 1.639606],accel_mss,speed_ms,0,blend_radius_m)
    movel([0.068472, -1.300176, -2.623010, -0.789204, 1.570796, 1.639268],accel_mss,speed_ms,0,blend_radius_m)
    movel([0.068228, -1.300130, -2.623037, -0.789222, 1.570796, 1.639025],accel_mss,speed_ms,0,blend_radius_m)
    movel([0.068160, -1.299903, -2.623172, -0.789314, 1.570796, 1.638957],accel_mss,speed_ms,0,blend_radius_m)
    movel([0.067957, -1.299756, -2.623260, -0.789373, 1.570796, 1.638753],accel_mss,speed_ms,0,blend_radius_m)
    movel([0.067920, -1.299501, -2.623411, -0.789476, 1.570796, 1.638717],accel_mss,speed_ms,0,blend_radius_m)
    movel([0.068076, -1.299095, -2.623653, -0.789641, 1.570796, 1.638872],accel_mss,speed_ms,0,blend_radius_m)
    movel([0.068245, -1.298825, -2.623814, -0.789750, 1.570796, 1.639041],accel_mss,speed_ms,0,blend_radius_m)
    movel([0.068538, -1.298372, -2.624083, -0.789934, 1.570796, 1.639334],accel_mss,speed_ms,0,blend_radius_m)
    movel([0.068564, -1.298071, -2.624261, -0.790056, 1.570796, 1.639361],accel_mss,speed_ms,0,blend_radius_m)
    movel([0.068351, -1.297911, -2.624356, -0.790122, 1.570796, 1.639147],accel_mss,speed_ms,0,blend_radius_m)
    movel([0.068159, -1.297750, -2.624452, -0.790187, 1.570796, 1.638955],accel_mss,speed_ms,0,blend_radius_m)
    movel([0.068070, -1.297551, -2.624570, -0.790268, 1.570796, 1.638866],accel_mss,speed_ms,0,blend_radius_m)
    movel([0.067838, -1.297444, -2.624633, -0.790312, 1.570796, 1.638635],accel_mss,speed_ms,0,blend_radius_m)
    movel([0.067733, -1.297246, -2.624751, -0.790392, 1.570796, 1.638529],accel_mss,speed_ms,0,blend_radius_m)
    movel([0.067965, -1.296990, -2.624902, -0.790497, 1.570796, 1.638762],accel_mss,speed_ms,0,blend_radius_m)
    movel([0.068177, -1.297285, -2.624727, -0.790376, 1.570796, 1.638973],accel_mss,speed_ms,0,blend_radius_m)
    movel([0.068448, -1.297463, -2.624622, -0.790304, 1.570796, 1.639244],accel_mss,speed_ms,0,blend_radius_m)
    movel([0.068582, -1.297195, -2.624781, -0.790413, 1.570796, 1.639379],accel_mss,speed_ms,0,blend_radius_m)
    movel([0.068570, -1.296945, -2.624929, -0.790515, 1.570796, 1.639366],accel_mss,speed_ms,0,blend_radius_m)
    movel([0.068283, -1.297098, -2.624839, -0.790453, 1.570796, 1.639079],accel_mss,speed_ms,0,blend_radius_m)
    movel([0.068322, -1.296834, -2.624995, -0.790560, 1.570796, 1.639119],accel_mss,speed_ms,0,blend_radius_m)
    movel([0.068410, -1.296575, -2.625148, -0.790666, 1.570796, 1.639206],accel_mss,speed_ms,0,blend_radius_m)
    movel([0.068413, -1.296331, -2.625292, -0.790766, 1.570796, 1.639209],accel_mss,speed_ms,0,blend_radius_m)
    movel([0.068610, -1.296024, -2.625474, -0.790891, 1.570796, 1.639406],accel_mss,speed_ms,0,blend_radius_m)
    movel([0.068344, -1.296042, -2.625463, -0.790884, 1.570796, 1.639140],accel_mss,speed_ms,0,blend_radius_m)
    movel([0.068247, -1.296349, -2.625281, -0.790758, 1.570796, 1.639043],accel_mss,speed_ms,0,blend_radius_m)
    movel([0.068015, -1.296285, -2.625319, -0.790785, 1.570796, 1.638811],accel_mss,speed_ms,0,blend_radius_m)
    movel([0.068098, -1.295843, -2.625580, -0.790965, 1.570796, 1.638894],accel_mss,speed_ms,0,blend_radius_m)
    movel([0.068346, -1.295534, -2.625763, -0.791092, 1.570796, 1.639142],accel_mss,speed_ms,0,blend_radius_m)
    movel([0.068703, -1.295215, -2.625951, -0.791223, 1.570796, 1.639499],accel_mss,speed_ms,0,blend_radius_m)
    movel([0.069005, -1.294904, -2.626135, -0.791351, 1.570796, 1.639802],accel_mss,speed_ms,0,blend_radius_m)
    movel([0.068736, -1.294446, -2.626405, -0.791539, 1.570796, 1.639533],accel_mss,speed_ms,0,blend_radius_m)
    movel([0.068447, -1.294179, -2.626561, -0.791649, 1.570796, 1.639243],accel_mss,speed_ms,0,blend_radius_m)
    movel([0.068186, -1.293987, -2.626674, -0.791727, 1.570796, 1.638982],accel_mss,speed_ms,0,blend_radius_m)
    movel([0.068055, -1.293698, -2.626844, -0.791847, 1.570796, 1.638851],accel_mss,speed_ms,0,blend_radius_m)
    movel([0.068400, -1.293396, -2.627022, -0.791971, 1.570796, 1.639196],accel_mss,speed_ms,0,blend_radius_m)
    movel([0.068673, -1.293222, -2.627124, -0.792043, 1.570796, 1.639470],accel_mss,speed_ms,0,blend_radius_m)
    movel([0.068591, -1.292993, -2.627259, -0.792138, 1.570796, 1.639387],accel_mss,speed_ms,0,blend_radius_m)
    movel([0.068494, -1.292776, -2.627386, -0.792227, 1.570796, 1.639291],accel_mss,speed_ms,0,blend_radius_m)
    movel([0.068508, -1.292532, -2.627529, -0.792328, 1.570796, 1.639305],accel_mss,speed_ms,0,blend_radius_m)
    movel([0.068313, -1.292435, -2.627586, -0.792368, 1.570796, 1.639109],accel_mss,speed_ms,0,blend_radius_m)
    movel([0.068432, -1.292054, -2.627809, -0.792526, 1.570796, 1.639228],accel_mss,speed_ms,0,blend_radius_m)
    movel([0.068734, -1.291591, -2.628080, -0.792718, 1.570796, 1.639530],accel_mss,speed_ms,0,blend_radius_m)
    movel([0.069080, -1.291360, -2.628215, -0.792814, 1.570796, 1.639876],accel_mss,speed_ms,0,blend_radius_m)
    movel([0.069351, -1.291183, -2.628319, -0.792887, 1.570796, 1.640148],accel_mss,speed_ms,0,blend_radius_m)
    movel([0.069675, -1.290933, -2.628465, -0.792991, 1.570796, 1.640471],accel_mss,speed_ms,0,blend_radius_m)
    movel([0.069973, -1.290833, -2.628523, -0.793033, 1.570796, 1.640769],accel_mss,speed_ms,0,blend_radius_m)
    movel([0.070329, -1.290548, -2.628690, -0.793151, 1.570796, 1.641125],accel_mss,speed_ms,0,blend_radius_m)
    movel([0.070734, -1.290402, -2.628775, -0.793212, 1.570796, 1.641530],accel_mss,speed_ms,0,blend_radius_m)
    movel([0.070848, -1.290597, -2.628661, -0.793131, 1.570796, 1.641644],accel_mss,speed_ms,0,blend_radius_m)
    movel([0.070586, -1.290557, -2.628684, -0.793148, 1.570796, 1.641382],accel_mss,speed_ms,0,blend_radius_m)
    movel([0.070545, -1.290828, -2.628526, -0.793035, 1.570796, 1.641341],accel_mss,speed_ms,0,blend_radius_m)
    movel([0.070287, -1.290805, -2.628540, -0.793044, 1.570796, 1.641083],accel_mss,speed_ms,0,blend_radius_m)
    movel([0.070092, -1.291071, -2.628384, -0.792934, 1.570796, 1.640888],accel_mss,speed_ms,0,blend_radius_m)
    movel([0.069788, -1.291216, -2.628299, -0.792873, 1.570796, 1.640584],accel_mss,speed_ms,0,blend_radius_m)
    movel([0.070023, -1.291249, -2.628280, -0.792860, 1.570796, 1.640820],accel_mss,speed_ms,0,blend_radius_m)
    movel([0.070448, -1.291024, -2.628412, -0.792954, 1.570796, 1.641244],accel_mss,speed_ms,0,blend_radius_m)
    movel([0.070733, -1.290883, -2.628494, -0.793012, 1.570796, 1.641529],accel_mss,speed_ms,0,blend_radius_m)
    movel([0.071014, -1.290753, -2.628570, -0.793066, 1.570796, 1.641811],accel_mss,speed_ms,0,blend_radius_m)
    movel([0.071419, -1.290544, -2.628692, -0.793153, 1.570796, 1.642215],accel_mss,speed_ms,0,blend_radius_m)
    movel([0.071699, -1.290195, -2.628896, -0.793298, 1.570796, 1.642496],accel_mss,speed_ms,0,blend_radius_m)
    movel([0.071397, -1.290344, -2.628808, -0.793236, 1.570796, 1.642193],accel_mss,speed_ms,0,blend_radius_m)
    movel([0.071394, -1.290015, -2.629001, -0.793373, 1.570796, 1.642190],accel_mss,speed_ms,0,blend_radius_m)
    movel([0.071674, -1.289807, -2.629122, -0.793460, 1.570796, 1.642471],accel_mss,speed_ms,0,blend_radius_m)
    movel([0.072099, -1.289622, -2.629230, -0.793537, 1.570796, 1.642895],accel_mss,speed_ms,0,blend_radius_m)
    movel([0.072618, -1.289439, -2.629336, -0.793614, 1.570796, 1.643415],accel_mss,speed_ms,0,blend_radius_m)
    movel([0.072298, -1.289775, -2.629140, -0.793473, 1.570796, 1.643094],accel_mss,speed_ms,0,blend_radius_m)
    movel([0.072072, -1.290052, -2.628979, -0.793358, 1.570796, 1.642868],accel_mss,speed_ms,0,blend_radius_m)
    movel([0.072318, -1.290082, -2.628962, -0.793345, 1.570796, 1.643115],accel_mss,speed_ms,0,blend_radius_m)
    movel([0.072810, -1.289907, -2.629064, -0.793418, 1.570796, 1.643606],accel_mss,speed_ms,0,blend_radius_m)
    movel([0.073098, -1.289924, -2.629053, -0.793411, 1.570796, 1.643895],accel_mss,speed_ms,0,blend_radius_m)
    movel([0.073371, -1.289879, -2.629080, -0.793430, 1.570796, 1.644167],accel_mss,speed_ms,0,blend_radius_m)
    movel([0.073643, -1.289667, -2.629204, -0.793519, 1.570796, 1.644439],accel_mss,speed_ms,0,blend_radius_m)
    movel([0.073422, -1.289556, -2.629268, -0.793565, 1.570796, 1.644218],accel_mss,speed_ms,0,blend_radius_m)
    movel([0.073605, -1.289116, -2.629525, -0.793749, 1.570796, 1.644402],accel_mss,speed_ms,0,blend_radius_m)
    movel([0.074088, -1.288858, -2.629674, -0.793857, 1.570796, 1.644884],accel_mss,speed_ms,0,blend_radius_m)
    movel([0.074586, -1.288774, -2.629723, -0.793892, 1.570796, 1.645382],accel_mss,speed_ms,0,blend_radius_m)
    movel([0.075419, -1.288701, -2.629765, -0.793922, 1.570796, 1.646216],accel_mss,speed_ms,0,blend_radius_m)
    movel([0.075774, -1.288673, -2.629782, -0.793934, 1.570796, 1.646570],accel_mss,speed_ms,0,blend_radius_m)
    movel([0.076162, -1.288635, -2.629804, -0.793950, 1.570796, 1.646959],accel_mss,speed_ms,0,blend_radius_m)
    movel([0.076529, -1.288597, -2.629826, -0.793966, 1.570796, 1.647325],accel_mss,speed_ms,0,blend_radius_m)
    movel([0.076800, -1.288565, -2.629845, -0.793979, 1.570796, 1.647596],accel_mss,speed_ms,0,blend_radius_m)
    movel([0.077294, -1.288560, -2.629848, -0.793981, 1.570796, 1.648090],accel_mss,speed_ms,0,blend_radius_m)
    movel([0.077690, -1.288646, -2.629798, -0.793945, 1.570796, 1.648486],accel_mss,speed_ms,0,blend_radius_m)
    movel([0.078122, -1.288841, -2.629684, -0.793864, 1.570796, 1.648918],accel_mss,speed_ms,0,blend_radius_m)
    movel([0.078432, -1.288951, -2.629621, -0.793818, 1.570796, 1.649228],accel_mss,speed_ms,0,blend_radius_m)
    movel([0.078708, -1.289007, -2.629588, -0.793794, 1.570796, 1.649504],accel_mss,speed_ms,0,blend_radius_m)
    movel([0.079022, -1.289032, -2.629573, -0.793784, 1.570796, 1.649819],accel_mss,speed_ms,0,blend_radius_m)
    movel([0.079477, -1.289125, -2.629519, -0.793745, 1.570796, 1.650273],accel_mss,speed_ms,0,blend_radius_m)
    movel([0.080017, -1.289405, -2.629356, -0.793628, 1.570796, 1.650813],accel_mss,speed_ms,0,blend_radius_m)
    movel([0.080490, -1.289761, -2.629149, -0.793479, 1.570796, 1.651286],accel_mss,speed_ms,0,blend_radius_m)
    movel([0.080723, -1.290104, -2.628949, -0.793336, 1.570796, 1.651519],accel_mss,speed_ms,0,blend_radius_m)
    movel([0.080790, -1.290461, -2.628740, -0.793187, 1.570796, 1.651586],accel_mss,speed_ms,0,blend_radius_m)
    movel([0.080755, -1.290906, -2.628480, -0.793002, 1.570796, 1.651551],accel_mss,speed_ms,0,blend_radius_m)
    movel([0.080623, -1.291367, -2.628211, -0.792811, 1.570796, 1.651420],accel_mss,speed_ms,0,blend_radius_m)
    movel([0.080414, -1.291769, -2.627976, -0.792644, 1.570796, 1.651210],accel_mss,speed_ms,0,blend_radius_m)
    movel([0.080193, -1.292059, -2.627806, -0.792524, 1.570796, 1.650990],accel_mss,speed_ms,0,blend_radius_m)
    movel([0.079916, -1.292349, -2.627636, -0.792404, 1.570796, 1.650712],accel_mss,speed_ms,0,blend_radius_m)
    movel([0.079600, -1.292623, -2.627475, -0.792290, 1.570796, 1.650396],accel_mss,speed_ms,0,blend_radius_m)
    movel([0.079260, -1.292868, -2.627332, -0.792189, 1.570796, 1.650056],accel_mss,speed_ms,0,blend_radius_m)
    movel([0.079132, -1.292699, -2.627431, -0.792259, 1.570796, 1.649929],accel_mss,speed_ms,0,blend_radius_m)
    movel([0.078790, -1.293064, -2.627217, -0.792108, 1.570796, 1.649586],accel_mss,speed_ms,0,blend_radius_m)
    movel([0.078548, -1.293294, -2.627082, -0.792013, 1.570796, 1.649345],accel_mss,speed_ms,0,blend_radius_m)
    movel([0.078210, -1.293734, -2.626823, -0.791832, 1.570796, 1.649006],accel_mss,speed_ms,0,blend_radius_m)
    movel([0.078166, -1.294015, -2.626658, -0.791716, 1.570796, 1.648962],accel_mss,speed_ms,0,blend_radius_m)
    movel([0.078357, -1.294349, -2.626462, -0.791579, 1.570796, 1.649153],accel_mss,speed_ms,0,blend_radius_m)
    movel([0.078391, -1.294602, -2.626313, -0.791475, 1.570796, 1.649187],accel_mss,speed_ms,0,blend_radius_m)
    movel([0.078328, -1.294883, -2.626147, -0.791359, 1.570796, 1.649124],accel_mss,speed_ms,0,blend_radius_m)
    movel([0.078048, -1.295310, -2.625895, -0.791184, 1.570796, 1.648844],accel_mss,speed_ms,0,blend_radius_m)
    movel([0.078070, -1.295548, -2.625754, -0.791086, 1.570796, 1.648866],accel_mss,speed_ms,0,blend_radius_m)
    movel([0.077797, -1.295930, -2.625529, -0.790930, 1.570796, 1.648593],accel_mss,speed_ms,0,blend_radius_m)
    movel([0.077543, -1.296213, -2.625362, -0.790814, 1.570796, 1.648340],accel_mss,speed_ms,0,blend_radius_m)
    movel([0.077141, -1.296453, -2.625220, -0.790716, 1.570796, 1.647937],accel_mss,speed_ms,0,blend_radius_m)
    movel([0.076881, -1.296662, -2.625096, -0.790630, 1.570796, 1.647677],accel_mss,speed_ms,0,blend_radius_m)
    movel([0.076380, -1.296832, -2.624996, -0.790561, 1.570796, 1.647176],accel_mss,speed_ms,0,blend_radius_m)
    movel([0.076038, -1.297953, -2.624332, -0.790105, 1.570796, 1.646834],accel_mss,speed_ms,0,blend_radius_m)
    movel([0.075953, -1.298382, -2.624077, -0.789930, 1.570796, 1.646749],accel_mss,speed_ms,0,blend_radius_m)
    movel([0.075814, -1.298681, -2.623899, -0.789809, 1.570796, 1.646610],accel_mss,speed_ms,0,blend_radius_m)
    movel([0.075570, -1.298998, -2.623711, -0.789680, 1.570796, 1.646366],accel_mss,speed_ms,0,blend_radius_m)
    movel([0.075189, -1.299340, -2.623508, -0.789542, 1.570796, 1.645986],accel_mss,speed_ms,0,blend_radius_m)
    movel([0.074854, -1.299474, -2.623428, -0.789487, 1.570796, 1.645650],accel_mss,speed_ms,0,blend_radius_m)
    movel([0.074612, -1.299705, -2.623290, -0.789394, 1.570796, 1.645408],accel_mss,speed_ms,0,blend_radius_m)
    movel([0.074370, -1.299617, -2.623343, -0.789430, 1.570796, 1.645166],accel_mss,speed_ms,0,blend_radius_m)
    movel([0.074338, -1.299900, -2.623174, -0.789315, 1.570796, 1.645134],accel_mss,speed_ms,0,blend_radius_m)
    movel([0.073982, -1.300051, -2.623084, -0.789254, 1.570796, 1.644779],accel_mss,speed_ms,0,blend_radius_m)
    speed_ms = 0.003
    movel([0.073982, -1.303545, -2.624704, -0.784140, 1.570796, 1.644779],accel_mss,speed_ms,0,blend_radius_m)
    speed_ms = 0.007
    movel([0.073932, -1.303284, -2.624861, -0.784245, 1.570796, 1.644728],accel_mss,speed_ms,0,blend_radius_m)
    movel([0.074261, -1.303044, -2.625004, -0.784341, 1.570796, 1.645057],accel_mss,speed_ms,0,blend_radius_m)
    movel([0.074673, -1.302820, -2.625138, -0.784431, 1.570796, 1.645470],accel_mss,speed_ms,0,blend_radius_m)
    movel([0.074331, -1.302852, -2.625119, -0.784418, 1.570796, 1.645127],accel_mss,speed_ms,0,blend_radius_m)
    movel([0.073782, -1.303089, -2.624977, -0.784323, 1.570796, 1.644579],accel_mss,speed_ms,0,blend_radius_m)
    movel([0.072985, -1.303366, -2.624811, -0.784211, 1.570796, 1.643781],accel_mss,speed_ms,0,blend_radius_m)
    movel([0.072179, -1.303619, -2.624660, -0.784110, 1.570796, 1.642975],accel_mss,speed_ms,0,blend_radius_m)
    movel([0.071902, -1.303597, -2.624673, -0.784119, 1.570796, 1.642698],accel_mss,speed_ms,0,blend_radius_m)
    movel([0.071682, -1.303891, -2.624497, -0.784001, 1.570796, 1.642478],accel_mss,speed_ms,0,blend_radius_m)
    movel([0.071302, -1.304085, -2.624380, -0.783923, 1.570796, 1.642098],accel_mss,speed_ms,0,blend_radius_m)
    movel([0.071480, -1.303802, -2.624551, -0.784037, 1.570796, 1.642277],accel_mss,speed_ms,0,blend_radius_m)
    movel([0.071194, -1.303858, -2.624517, -0.784014, 1.570796, 1.641991],accel_mss,speed_ms,0,blend_radius_m)
    movel([0.070917, -1.304036, -2.624410, -0.783943, 1.570796, 1.641714],accel_mss,speed_ms,0,blend_radius_m)
    movel([0.070724, -1.303876, -2.624506, -0.784007, 1.570796, 1.641520],accel_mss,speed_ms,0,blend_radius_m)
    movel([0.070555, -1.303705, -2.624608, -0.784075, 1.570796, 1.641352],accel_mss,speed_ms,0,blend_radius_m)
    movel([0.070266, -1.303698, -2.624613, -0.784078, 1.570796, 1.641063],accel_mss,speed_ms,0,blend_radius_m)
    movel([0.070498, -1.303789, -2.624558, -0.784042, 1.570796, 1.641294],accel_mss,speed_ms,0,blend_radius_m)
    movel([0.070207, -1.303999, -2.624432, -0.783958, 1.570796, 1.641004],accel_mss,speed_ms,0,blend_radius_m)
    movel([0.069999, -1.303927, -2.624476, -0.783987, 1.570796, 1.640795],accel_mss,speed_ms,0,blend_radius_m)
    movel([0.069864, -1.303770, -2.624569, -0.784049, 1.570796, 1.640660],accel_mss,speed_ms,0,blend_radius_m)
    movel([0.069616, -1.303985, -2.624441, -0.783964, 1.570796, 1.640412],accel_mss,speed_ms,0,blend_radius_m)
    movel([0.069394, -1.303915, -2.624483, -0.783992, 1.570796, 1.640190],accel_mss,speed_ms,0,blend_radius_m)
    movel([0.069164, -1.303567, -2.624691, -0.784131, 1.570796, 1.639960],accel_mss,speed_ms,0,blend_radius_m)
    movel([0.068809, -1.303606, -2.624668, -0.784115, 1.570796, 1.639606],accel_mss,speed_ms,0,blend_radius_m)
    movel([0.068472, -1.303670, -2.624630, -0.784090, 1.570796, 1.639268],accel_mss,speed_ms,0,blend_radius_m)
    movel([0.068228, -1.303624, -2.624657, -0.784108, 1.570796, 1.639025],accel_mss,speed_ms,0,blend_radius_m)
    movel([0.068160, -1.303397, -2.624793, -0.784199, 1.570796, 1.638957],accel_mss,speed_ms,0,blend_radius_m)
    movel([0.067957, -1.303250, -2.624881, -0.784258, 1.570796, 1.638753],accel_mss,speed_ms,0,blend_radius_m)
    movel([0.067920, -1.302997, -2.625033, -0.784360, 1.570796, 1.638717],accel_mss,speed_ms,0,blend_radius_m)
    movel([0.068076, -1.302591, -2.625275, -0.784523, 1.570796, 1.638872],accel_mss,speed_ms,0,blend_radius_m)
    movel([0.068245, -1.302321, -2.625436, -0.784631, 1.570796, 1.639041],accel_mss,speed_ms,0,blend_radius_m)
    movel([0.068538, -1.301870, -2.625706, -0.784813, 1.570796, 1.639334],accel_mss,speed_ms,0,blend_radius_m)
    movel([0.068564, -1.301570, -2.625885, -0.784934, 1.570796, 1.639361],accel_mss,speed_ms,0,blend_radius_m)
    movel([0.068351, -1.301410, -2.625980, -0.784999, 1.570796, 1.639147],accel_mss,speed_ms,0,blend_radius_m)
    movel([0.068159, -1.301249, -2.626076, -0.785063, 1.570796, 1.638955],accel_mss,speed_ms,0,blend_radius_m)
    movel([0.068070, -1.301051, -2.626194, -0.785144, 1.570796, 1.638866],accel_mss,speed_ms,0,blend_radius_m)
    movel([0.067838, -1.300944, -2.626258, -0.785187, 1.570796, 1.638635],accel_mss,speed_ms,0,blend_radius_m)
    movel([0.067733, -1.300746, -2.626376, -0.785267, 1.570796, 1.638529],accel_mss,speed_ms,0,blend_radius_m)
    movel([0.067965, -1.300491, -2.626528, -0.785370, 1.570796, 1.638762],accel_mss,speed_ms,0,blend_radius_m)
    movel([0.068177, -1.300786, -2.626352, -0.785251, 1.570796, 1.638973],accel_mss,speed_ms,0,blend_radius_m)
    movel([0.068448, -1.300963, -2.626247, -0.785179, 1.570796, 1.639244],accel_mss,speed_ms,0,blend_radius_m)
    movel([0.068582, -1.300695, -2.626406, -0.785288, 1.570796, 1.639379],accel_mss,speed_ms,0,blend_radius_m)
    movel([0.068570, -1.300446, -2.626554, -0.785388, 1.570796, 1.639366],accel_mss,speed_ms,0,blend_radius_m)
    movel([0.068283, -1.300598, -2.626464, -0.785327, 1.570796, 1.639079],accel_mss,speed_ms,0,blend_radius_m)
    movel([0.068322, -1.300335, -2.626620, -0.785433, 1.570796, 1.639119],accel_mss,speed_ms,0,blend_radius_m)
    movel([0.068410, -1.300077, -2.626774, -0.785538, 1.570796, 1.639206],accel_mss,speed_ms,0,blend_radius_m)
    movel([0.068413, -1.299834, -2.626919, -0.785637, 1.570796, 1.639209],accel_mss,speed_ms,0,blend_radius_m)
    movel([0.068610, -1.299527, -2.627101, -0.785761, 1.570796, 1.639406],accel_mss,speed_ms,0,blend_radius_m)
    movel([0.068344, -1.299545, -2.627090, -0.785754, 1.570796, 1.639140],accel_mss,speed_ms,0,blend_radius_m)
    movel([0.068247, -1.299852, -2.626908, -0.785629, 1.570796, 1.639043],accel_mss,speed_ms,0,blend_radius_m)
    movel([0.068015, -1.299788, -2.626946, -0.785655, 1.570796, 1.638811],accel_mss,speed_ms,0,blend_radius_m)
    movel([0.068098, -1.299347, -2.627208, -0.785834, 1.570796, 1.638894],accel_mss,speed_ms,0,blend_radius_m)
    movel([0.068346, -1.299039, -2.627391, -0.785960, 1.570796, 1.639142],accel_mss,speed_ms,0,blend_radius_m)
    movel([0.068703, -1.298720, -2.627579, -0.786089, 1.570796, 1.639499],accel_mss,speed_ms,0,blend_radius_m)
    movel([0.069005, -1.298409, -2.627764, -0.786216, 1.570796, 1.639802],accel_mss,speed_ms,0,blend_radius_m)
    movel([0.068736, -1.297952, -2.628034, -0.786402, 1.570796, 1.639533],accel_mss,speed_ms,0,blend_radius_m)
    movel([0.068447, -1.297686, -2.628192, -0.786511, 1.570796, 1.639243],accel_mss,speed_ms,0,blend_radius_m)
    movel([0.068186, -1.297495, -2.628305, -0.786589, 1.570796, 1.638982],accel_mss,speed_ms,0,blend_radius_m)
    movel([0.068055, -1.297206, -2.628475, -0.786707, 1.570796, 1.638851],accel_mss,speed_ms,0,blend_radius_m)
    movel([0.068400, -1.296905, -2.628653, -0.786831, 1.570796, 1.639196],accel_mss,speed_ms,0,blend_radius_m)
    movel([0.068673, -1.296731, -2.628756, -0.786902, 1.570796, 1.639470],accel_mss,speed_ms,0,blend_radius_m)
    movel([0.068591, -1.296502, -2.628891, -0.786996, 1.570796, 1.639387],accel_mss,speed_ms,0,blend_radius_m)
    movel([0.068494, -1.296286, -2.629019, -0.787084, 1.570796, 1.639291],accel_mss,speed_ms,0,blend_radius_m)
    movel([0.068508, -1.296042, -2.629162, -0.787184, 1.570796, 1.639305],accel_mss,speed_ms,0,blend_radius_m)
    movel([0.068313, -1.295946, -2.629219, -0.787224, 1.570796, 1.639109],accel_mss,speed_ms,0,blend_radius_m)
    movel([0.068432, -1.295566, -2.629443, -0.787380, 1.570796, 1.639228],accel_mss,speed_ms,0,blend_radius_m)
    movel([0.068734, -1.295104, -2.629715, -0.787570, 1.570796, 1.639530],accel_mss,speed_ms,0,blend_radius_m)
    movel([0.069080, -1.294873, -2.629850, -0.787665, 1.570796, 1.639876],accel_mss,speed_ms,0,blend_radius_m)
    movel([0.069351, -1.294697, -2.629954, -0.787738, 1.570796, 1.640148],accel_mss,speed_ms,0,blend_radius_m)
    movel([0.069675, -1.294448, -2.630100, -0.787841, 1.570796, 1.640471],accel_mss,speed_ms,0,blend_radius_m)
    movel([0.069973, -1.294347, -2.630159, -0.787882, 1.570796, 1.640769],accel_mss,speed_ms,0,blend_radius_m)
    movel([0.070329, -1.294063, -2.630326, -0.788000, 1.570796, 1.641125],accel_mss,speed_ms,0,blend_radius_m)
    movel([0.070734, -1.293918, -2.630411, -0.788060, 1.570796, 1.641530],accel_mss,speed_ms,0,blend_radius_m)
    movel([0.070848, -1.294112, -2.630297, -0.787979, 1.570796, 1.641644],accel_mss,speed_ms,0,blend_radius_m)
    movel([0.070586, -1.294072, -2.630321, -0.787996, 1.570796, 1.641382],accel_mss,speed_ms,0,blend_radius_m)
    movel([0.070545, -1.294342, -2.630162, -0.787884, 1.570796, 1.641341],accel_mss,speed_ms,0,blend_radius_m)
    movel([0.070287, -1.294320, -2.630176, -0.787894, 1.570796, 1.641083],accel_mss,speed_ms,0,blend_radius_m)
    movel([0.070092, -1.294585, -2.630020, -0.787784, 1.570796, 1.640888],accel_mss,speed_ms,0,blend_radius_m)
    movel([0.069788, -1.294730, -2.629935, -0.787724, 1.570796, 1.640584],accel_mss,speed_ms,0,blend_radius_m)
    movel([0.070023, -1.294763, -2.629915, -0.787711, 1.570796, 1.640820],accel_mss,speed_ms,0,blend_radius_m)
    movel([0.070448, -1.294538, -2.630047, -0.787804, 1.570796, 1.641244],accel_mss,speed_ms,0,blend_radius_m)
    movel([0.070733, -1.294397, -2.630130, -0.787862, 1.570796, 1.641529],accel_mss,speed_ms,0,blend_radius_m)
    movel([0.071014, -1.294267, -2.630206, -0.787915, 1.570796, 1.641811],accel_mss,speed_ms,0,blend_radius_m)
    movel([0.071419, -1.294059, -2.630329, -0.788002, 1.570796, 1.642215],accel_mss,speed_ms,0,blend_radius_m)
    movel([0.071699, -1.293711, -2.630533, -0.788145, 1.570796, 1.642496],accel_mss,speed_ms,0,blend_radius_m)
    movel([0.071397, -1.293860, -2.630445, -0.788084, 1.570796, 1.642193],accel_mss,speed_ms,0,blend_radius_m)
    movel([0.071394, -1.293531, -2.630638, -0.788220, 1.570796, 1.642190],accel_mss,speed_ms,0,blend_radius_m)
    movel([0.071674, -1.293324, -2.630760, -0.788306, 1.570796, 1.642471],accel_mss,speed_ms,0,blend_radius_m)
    movel([0.072099, -1.293139, -2.630868, -0.788382, 1.570796, 1.642895],accel_mss,speed_ms,0,blend_radius_m)
    movel([0.072618, -1.292956, -2.630975, -0.788458, 1.570796, 1.643415],accel_mss,speed_ms,0,blend_radius_m)
    movel([0.072298, -1.293292, -2.630778, -0.788319, 1.570796, 1.643094],accel_mss,speed_ms,0,blend_radius_m)
    movel([0.072072, -1.293569, -2.630616, -0.788204, 1.570796, 1.642868],accel_mss,speed_ms,0,blend_radius_m)
    movel([0.072318, -1.293598, -2.630599, -0.788192, 1.570796, 1.643115],accel_mss,speed_ms,0,blend_radius_m)
    movel([0.072810, -1.293423, -2.630701, -0.788264, 1.570796, 1.643606],accel_mss,speed_ms,0,blend_radius_m)
    movel([0.073098, -1.293441, -2.630691, -0.788257, 1.570796, 1.643895],accel_mss,speed_ms,0,blend_radius_m)
    movel([0.073371, -1.293396, -2.630718, -0.788276, 1.570796, 1.644167],accel_mss,speed_ms,0,blend_radius_m)
    movel([0.073643, -1.293184, -2.630842, -0.788364, 1.570796, 1.644439],accel_mss,speed_ms,0,blend_radius_m)
    movel([0.073422, -1.293074, -2.630906, -0.788409, 1.570796, 1.644218],accel_mss,speed_ms,0,blend_radius_m)
    movel([0.073605, -1.292634, -2.631163, -0.788592, 1.570796, 1.644402],accel_mss,speed_ms,0,blend_radius_m)
    movel([0.074088, -1.292377, -2.631314, -0.788698, 1.570796, 1.644884],accel_mss,speed_ms,0,blend_radius_m)
    movel([0.074586, -1.292293, -2.631363, -0.788733, 1.570796, 1.645382],accel_mss,speed_ms,0,blend_radius_m)
    movel([0.075419, -1.292221, -2.631405, -0.788763, 1.570796, 1.646216],accel_mss,speed_ms,0,blend_radius_m)
    movel([0.075774, -1.292192, -2.631422, -0.788775, 1.570796, 1.646570],accel_mss,speed_ms,0,blend_radius_m)
    movel([0.076162, -1.292154, -2.631444, -0.788791, 1.570796, 1.646959],accel_mss,speed_ms,0,blend_radius_m)
    movel([0.076529, -1.292117, -2.631466, -0.788806, 1.570796, 1.647325],accel_mss,speed_ms,0,blend_radius_m)
    movel([0.076800, -1.292084, -2.631485, -0.788820, 1.570796, 1.647596],accel_mss,speed_ms,0,blend_radius_m)
    movel([0.077294, -1.292079, -2.631488, -0.788822, 1.570796, 1.648090],accel_mss,speed_ms,0,blend_radius_m)
    movel([0.077690, -1.292165, -2.631437, -0.788786, 1.570796, 1.648486],accel_mss,speed_ms,0,blend_radius_m)
    movel([0.078122, -1.292360, -2.631324, -0.788705, 1.570796, 1.648918],accel_mss,speed_ms,0,blend_radius_m)
    movel([0.078432, -1.292469, -2.631260, -0.788660, 1.570796, 1.649228],accel_mss,speed_ms,0,blend_radius_m)
    movel([0.078708, -1.292526, -2.631227, -0.788636, 1.570796, 1.649504],accel_mss,speed_ms,0,blend_radius_m)
    movel([0.079022, -1.292550, -2.631212, -0.788626, 1.570796, 1.649819],accel_mss,speed_ms,0,blend_radius_m)
    movel([0.079477, -1.292643, -2.631158, -0.788588, 1.570796, 1.650273],accel_mss,speed_ms,0,blend_radius_m)
    movel([0.080017, -1.292922, -2.630995, -0.788472, 1.570796, 1.650813],accel_mss,speed_ms,0,blend_radius_m)
    movel([0.080490, -1.293278, -2.630787, -0.788325, 1.570796, 1.651286],accel_mss,speed_ms,0,blend_radius_m)
    movel([0.080723, -1.293620, -2.630586, -0.788183, 1.570796, 1.651519],accel_mss,speed_ms,0,blend_radius_m)
    movel([0.080790, -1.293977, -2.630377, -0.788035, 1.570796, 1.651586],accel_mss,speed_ms,0,blend_radius_m)
    movel([0.080755, -1.294421, -2.630116, -0.787852, 1.570796, 1.651551],accel_mss,speed_ms,0,blend_radius_m)
    movel([0.080623, -1.294881, -2.629846, -0.787662, 1.570796, 1.651420],accel_mss,speed_ms,0,blend_radius_m)
    movel([0.080414, -1.295282, -2.629610, -0.787497, 1.570796, 1.651210],accel_mss,speed_ms,0,blend_radius_m)
    movel([0.080193, -1.295571, -2.629440, -0.787378, 1.570796, 1.650990],accel_mss,speed_ms,0,blend_radius_m)
    movel([0.079916, -1.295860, -2.629270, -0.787259, 1.570796, 1.650712],accel_mss,speed_ms,0,blend_radius_m)
    movel([0.079600, -1.296134, -2.629108, -0.787147, 1.570796, 1.650396],accel_mss,speed_ms,0,blend_radius_m)
    movel([0.079260, -1.296379, -2.628964, -0.787046, 1.570796, 1.650056],accel_mss,speed_ms,0,blend_radius_m)
    movel([0.079132, -1.296209, -2.629064, -0.787116, 1.570796, 1.649929],accel_mss,speed_ms,0,blend_radius_m)
    movel([0.078790, -1.296573, -2.628849, -0.786967, 1.570796, 1.649586],accel_mss,speed_ms,0,blend_radius_m)
    movel([0.078548, -1.296803, -2.628714, -0.786872, 1.570796, 1.649345],accel_mss,speed_ms,0,blend_radius_m)
    movel([0.078210, -1.297243, -2.628454, -0.786692, 1.570796, 1.649006],accel_mss,speed_ms,0,blend_radius_m)
    movel([0.078166, -1.297522, -2.628289, -0.786578, 1.570796, 1.648962],accel_mss,speed_ms,0,blend_radius_m)
    movel([0.078357, -1.297855, -2.628092, -0.786442, 1.570796, 1.649153],accel_mss,speed_ms,0,blend_radius_m)
    movel([0.078391, -1.298108, -2.627942, -0.786339, 1.570796, 1.649187],accel_mss,speed_ms,0,blend_radius_m)
    movel([0.078328, -1.298389, -2.627776, -0.786224, 1.570796, 1.649124],accel_mss,speed_ms,0,blend_radius_m)
    movel([0.078048, -1.298815, -2.627523, -0.786051, 1.570796, 1.648844],accel_mss,speed_ms,0,blend_radius_m)
    movel([0.078070, -1.299052, -2.627382, -0.785954, 1.570796, 1.648866],accel_mss,speed_ms,0,blend_radius_m)
    movel([0.077797, -1.299433, -2.627156, -0.785799, 1.570796, 1.648593],accel_mss,speed_ms,0,blend_radius_m)
    movel([0.077543, -1.299716, -2.626989, -0.785685, 1.570796, 1.648340],accel_mss,speed_ms,0,blend_radius_m)
    movel([0.077141, -1.299955, -2.626847, -0.785588, 1.570796, 1.647937],accel_mss,speed_ms,0,blend_radius_m)
    movel([0.076881, -1.300164, -2.626722, -0.785503, 1.570796, 1.647677],accel_mss,speed_ms,0,blend_radius_m)
    movel([0.076380, -1.300334, -2.626621, -0.785434, 1.570796, 1.647176],accel_mss,speed_ms,0,blend_radius_m)
    movel([0.076038, -1.301452, -2.625956, -0.784982, 1.570796, 1.646834],accel_mss,speed_ms,0,blend_radius_m)
    movel([0.075953, -1.301880, -2.625700, -0.784809, 1.570796, 1.646749],accel_mss,speed_ms,0,blend_radius_m)
    movel([0.075814, -1.302178, -2.625522, -0.784689, 1.570796, 1.646610],accel_mss,speed_ms,0,blend_radius_m)
    movel([0.075570, -1.302494, -2.625333, -0.784562, 1.570796, 1.646366],accel_mss,speed_ms,0,blend_radius_m)
    movel([0.075189, -1.302835, -2.625129, -0.784425, 1.570796, 1.645986],accel_mss,speed_ms,0,blend_radius_m)
    movel([0.074854, -1.302969, -2.625049, -0.784371, 1.570796, 1.645650],accel_mss,speed_ms,0,blend_radius_m)
    movel([0.074612, -1.303200, -2.624911, -0.784278, 1.570796, 1.645408],accel_mss,speed_ms,0,blend_radius_m)
    movel([0.074370, -1.303112, -2.624964, -0.784313, 1.570796, 1.645166],accel_mss,speed_ms,0,blend_radius_m)
    movel([0.074338, -1.303394, -2.624794, -0.784200, 1.570796, 1.645134],accel_mss,speed_ms,0,blend_radius_m)
    movel([0.073982, -1.303545, -2.624704, -0.784140, 1.570796, 1.644779],accel_mss,speed_ms,0,blend_radius_m)
    speed_ms = 0.003
    movel([0.073982, -1.289735, -2.618173, -0.804481, 1.570796, 1.644779],accel_mss,speed_ms,0,blend_radius_m)
    speed_ms = 1.000
    movel([0.073982, -1.263429, -2.604724, -0.844235, 1.570796, 1.644779],accel_mss,speed_ms,0,blend_radius_m)
    movel([0.076909, -1.251042, -2.611644, -0.849703, 1.570796, 1.647706],accel_mss,speed_ms,0,blend_radius_m)
    movel([0.076909, -1.277513, -2.625256, -0.809620, 1.570796, 1.647706],accel_mss,speed_ms,0,blend_radius_m)
    speed_ms = 0.003
    movel([0.076909, -1.287904, -2.630229, -0.794256, 1.570796, 1.647706],accel_mss,speed_ms,0,blend_radius_m)
    speed_ms = 0.007
    movel([0.076129, -1.288050, -2.630144, -0.794195, 1.570796, 1.646925],accel_mss,speed_ms,0,blend_radius_m)
    movel([0.075299, -1.288083, -2.630125, -0.794181, 1.570796, 1.646095],accel_mss,speed_ms,0,blend_radius_m)
    movel([0.074609, -1.288022, -2.630160, -0.794207, 1.570796, 1.645406],accel_mss,speed_ms,0,blend_radius_m)
    movel([0.074509, -1.287833, -2.630270, -0.794286, 1.570796, 1.645305],accel_mss,speed_ms,0,blend_radius_m)
    movel([0.074808, -1.287539, -2.630440, -0.794409, 1.570796, 1.645604],accel_mss,speed_ms,0,blend_radius_m)
    movel([0.075762, -1.287303, -2.630578, -0.794509, 1.570796, 1.646558],accel_mss,speed_ms,0,blend_radius_m)
    movel([0.076791, -1.287181, -2.630648, -0.794560, 1.570796, 1.647587],accel_mss,speed_ms,0,blend_radius_m)
    movel([0.077546, -1.287262, -2.630601, -0.794526, 1.570796, 1.648343],accel_mss,speed_ms,0,blend_radius_m)
    movel([0.077806, -1.287388, -2.630528, -0.794473, 1.570796, 1.648603],accel_mss,speed_ms,0,blend_radius_m)
    movel([0.077509, -1.287716, -2.630338, -0.794335, 1.570796, 1.648305],accel_mss,speed_ms,0,blend_radius_m)
    movel([0.076909, -1.287904, -2.630229, -0.794256, 1.570796, 1.647706],accel_mss,speed_ms,0,blend_radius_m)
    speed_ms = 0.003
    movel([0.076909, -1.291425, -2.631870, -0.789094, 1.570796, 1.647706],accel_mss,speed_ms,0,blend_radius_m)
    speed_ms = 0.007
    movel([0.076129, -1.291571, -2.631785, -0.789034, 1.570796, 1.646925],accel_mss,speed_ms,0,blend_radius_m)
    movel([0.075299, -1.291604, -2.631765, -0.789020, 1.570796, 1.646095],accel_mss,speed_ms,0,blend_radius_m)
    movel([0.074609, -1.291543, -2.631801, -0.789045, 1.570796, 1.645406],accel_mss,speed_ms,0,blend_radius_m)
    movel([0.074509, -1.291354, -2.631911, -0.789124, 1.570796, 1.645305],accel_mss,speed_ms,0,blend_radius_m)
    movel([0.074808, -1.291061, -2.632082, -0.789246, 1.570796, 1.645604],accel_mss,speed_ms,0,blend_radius_m)
    movel([0.075762, -1.290825, -2.632220, -0.789345, 1.570796, 1.646558],accel_mss,speed_ms,0,blend_radius_m)
    movel([0.076791, -1.290704, -2.632290, -0.789395, 1.570796, 1.647587],accel_mss,speed_ms,0,blend_radius_m)
    movel([0.077546, -1.290784, -2.632243, -0.789362, 1.570796, 1.648343],accel_mss,speed_ms,0,blend_radius_m)
    movel([0.077806, -1.290910, -2.632170, -0.789309, 1.570796, 1.648603],accel_mss,speed_ms,0,blend_radius_m)
    movel([0.077509, -1.291238, -2.631979, -0.789172, 1.570796, 1.648305],accel_mss,speed_ms,0,blend_radius_m)
    movel([0.076909, -1.291425, -2.631870, -0.789094, 1.570796, 1.647706],accel_mss,speed_ms,0,blend_radius_m)
    speed_ms = 0.003
    movel([0.076909, -1.277513, -2.625256, -0.809620, 1.570796, 1.647706],accel_mss,speed_ms,0,blend_radius_m)
    speed_ms = 1.000
    movel([0.076909, -1.251042, -2.611644, -0.849703, 1.570796, 1.647706],accel_mss,speed_ms,0,blend_radius_m)
    movel([0.077291, -1.249693, -2.612387, -0.850309, 1.570796, 1.648088],accel_mss,speed_ms,0,blend_radius_m)
    movel([0.077291, -1.276182, -2.626016, -0.810191, 1.570796, 1.648088],accel_mss,speed_ms,0,blend_radius_m)
    speed_ms = 0.003
    movel([0.077291, -1.286581, -2.630996, -0.794812, 1.570796, 1.648088],accel_mss,speed_ms,0,blend_radius_m)
    speed_ms = 0.007
    movel([0.076492, -1.286619, -2.630974, -0.794796, 1.570796, 1.647288],accel_mss,speed_ms,0,blend_radius_m)
    movel([0.075702, -1.286738, -2.630905, -0.794746, 1.570796, 1.646499],accel_mss,speed_ms,0,blend_radius_m)
    movel([0.075018, -1.286926, -2.630796, -0.794667, 1.570796, 1.645814],accel_mss,speed_ms,0,blend_radius_m)
    movel([0.074481, -1.287038, -2.630731, -0.794620, 1.570796, 1.645277],accel_mss,speed_ms,0,blend_radius_m)
    movel([0.074238, -1.286897, -2.630813, -0.794680, 1.570796, 1.645034],accel_mss,speed_ms,0,blend_radius_m)
    movel([0.074188, -1.286422, -2.631088, -0.794880, 1.570796, 1.644984],accel_mss,speed_ms,0,blend_radius_m)
    movel([0.074355, -1.285032, -2.631890, -0.795466, 1.570796, 1.645151],accel_mss,speed_ms,0,blend_radius_m)
    movel([0.074579, -1.283540, -2.632750, -0.796099, 1.570796, 1.645376],accel_mss,speed_ms,0,blend_radius_m)
    movel([0.074809, -1.282447, -2.633377, -0.796565, 1.570796, 1.645605],accel_mss,speed_ms,0,blend_radius_m)
    movel([0.075052, -1.281644, -2.633838, -0.796908, 1.570796, 1.645848],accel_mss,speed_ms,0,blend_radius_m)
    movel([0.075328, -1.281134, -2.634129, -0.797126, 1.570796, 1.646124],accel_mss,speed_ms,0,blend_radius_m)
    movel([0.076329, -1.280304, -2.634603, -0.797481, 1.570796, 1.647126],accel_mss,speed_ms,0,blend_radius_m)
    movel([0.078074, -1.279627, -2.634990, -0.797772, 1.570796, 1.648871],accel_mss,speed_ms,0,blend_radius_m)
    movel([0.079946, -1.279261, -2.635198, -0.797930, 1.570796, 1.650742],accel_mss,speed_ms,0,blend_radius_m)
    movel([0.081399, -1.279367, -2.635138, -0.797884, 1.570796, 1.652195],accel_mss,speed_ms,0,blend_radius_m)
    movel([0.081937, -1.279667, -2.634967, -0.797755, 1.570796, 1.652733],accel_mss,speed_ms,0,blend_radius_m)
    movel([0.082153, -1.280164, -2.634683, -0.797542, 1.570796, 1.652949],accel_mss,speed_ms,0,blend_radius_m)
    movel([0.082056, -1.280944, -2.634238, -0.797207, 1.570796, 1.652852],accel_mss,speed_ms,0,blend_radius_m)
    movel([0.081621, -1.282158, -2.633543, -0.796688, 1.570796, 1.652417],accel_mss,speed_ms,0,blend_radius_m)
    movel([0.081209, -1.283020, -2.633048, -0.796320, 1.570796, 1.652006],accel_mss,speed_ms,0,blend_radius_m)
    movel([0.080540, -1.284202, -2.632369, -0.795818, 1.570796, 1.651337],accel_mss,speed_ms,0,blend_radius_m)
    movel([0.079825, -1.285365, -2.631699, -0.795326, 1.570796, 1.650622],accel_mss,speed_ms,0,blend_radius_m)
    movel([0.079256, -1.286161, -2.631238, -0.794989, 1.570796, 1.650053],accel_mss,speed_ms,0,blend_radius_m)
    movel([0.078803, -1.286738, -2.630905, -0.794746, 1.570796, 1.649599],accel_mss,speed_ms,0,blend_radius_m)
    movel([0.078012, -1.286628, -2.630968, -0.794793, 1.570796, 1.648808],accel_mss,speed_ms,0,blend_radius_m)
    movel([0.077291, -1.286581, -2.630996, -0.794812, 1.570796, 1.648088],accel_mss,speed_ms,0,blend_radius_m)
    speed_ms = 0.003
    movel([0.077291, -1.290105, -2.632639, -0.789645, 1.570796, 1.648088],accel_mss,speed_ms,0,blend_radius_m)
    speed_ms = 0.007
    movel([0.076492, -1.290143, -2.632617, -0.789630, 1.570796, 1.647288],accel_mss,speed_ms,0,blend_radius_m)
    movel([0.075702, -1.290262, -2.632548, -0.789580, 1.570796, 1.646499],accel_mss,speed_ms,0,blend_radius_m)
    movel([0.075018, -1.290449, -2.632439, -0.789502, 1.570796, 1.645814],accel_mss,speed_ms,0,blend_radius_m)
    movel([0.074481, -1.290561, -2.632373, -0.789455, 1.570796, 1.645277],accel_mss,speed_ms,0,blend_radius_m)
    movel([0.074238, -1.290420, -2.632456, -0.789514, 1.570796, 1.645034],accel_mss,speed_ms,0,blend_radius_m)
    movel([0.074188, -1.289946, -2.632731, -0.789712, 1.570796, 1.644984],accel_mss,speed_ms,0,blend_radius_m)
    movel([0.074355, -1.288559, -2.633536, -0.790293, 1.570796, 1.645151],accel_mss,speed_ms,0,blend_radius_m)
    movel([0.074579, -1.287070, -2.634398, -0.790921, 1.570796, 1.645376],accel_mss,speed_ms,0,blend_radius_m)
    movel([0.074809, -1.285980, -2.635028, -0.791382, 1.570796, 1.645605],accel_mss,speed_ms,0,blend_radius_m)
    movel([0.075052, -1.285178, -2.635489, -0.791722, 1.570796, 1.645848],accel_mss,speed_ms,0,blend_radius_m)
    movel([0.075328, -1.284669, -2.635782, -0.791938, 1.570796, 1.646124],accel_mss,speed_ms,0,blend_radius_m)
    movel([0.076329, -1.283841, -2.636257, -0.792290, 1.570796, 1.647126],accel_mss,speed_ms,0,blend_radius_m)
    movel([0.078074, -1.283166, -2.636645, -0.792579, 1.570796, 1.648871],accel_mss,speed_ms,0,blend_radius_m)
    movel([0.079946, -1.282800, -2.636854, -0.792735, 1.570796, 1.650742],accel_mss,speed_ms,0,blend_radius_m)
    movel([0.081399, -1.282906, -2.636793, -0.792689, 1.570796, 1.652195],accel_mss,speed_ms,0,blend_radius_m)
    movel([0.081937, -1.283206, -2.636622, -0.792562, 1.570796, 1.652733],accel_mss,speed_ms,0,blend_radius_m)
    movel([0.082153, -1.283701, -2.636338, -0.792350, 1.570796, 1.652949],accel_mss,speed_ms,0,blend_radius_m)
    movel([0.082056, -1.284479, -2.635891, -0.792019, 1.570796, 1.652852],accel_mss,speed_ms,0,blend_radius_m)
    movel([0.081621, -1.285691, -2.635194, -0.791504, 1.570796, 1.652417],accel_mss,speed_ms,0,blend_radius_m)
    movel([0.081209, -1.286552, -2.634698, -0.791140, 1.570796, 1.652006],accel_mss,speed_ms,0,blend_radius_m)
    movel([0.080540, -1.287731, -2.634016, -0.790642, 1.570796, 1.651337],accel_mss,speed_ms,0,blend_radius_m)
    movel([0.079825, -1.288891, -2.633344, -0.790154, 1.570796, 1.650622],accel_mss,speed_ms,0,blend_radius_m)
    movel([0.079256, -1.289686, -2.632882, -0.789821, 1.570796, 1.650053],accel_mss,speed_ms,0,blend_radius_m)
    movel([0.078803, -1.290261, -2.632548, -0.789580, 1.570796, 1.649599],accel_mss,speed_ms,0,blend_radius_m)
    movel([0.078012, -1.290152, -2.632611, -0.789626, 1.570796, 1.648808],accel_mss,speed_ms,0,blend_radius_m)
    movel([0.077291, -1.290105, -2.632639, -0.789645, 1.570796, 1.648088],accel_mss,speed_ms,0,blend_radius_m)
    speed_ms = 0.003
    movel([0.077291, -1.276182, -2.626016, -0.810191, 1.570796, 1.648088],accel_mss,speed_ms,0,blend_radius_m)
    speed_ms = 1.000
    movel([0.077291, -1.249693, -2.612387, -0.850309, 1.570796, 1.648088],accel_mss,speed_ms,0,blend_radius_m)
    movel([0.079543, -1.241590, -2.616802, -0.853997, 1.570796, 1.650339],accel_mss,speed_ms,0,blend_radius_m)
    movel([0.079543, -1.268182, -2.630539, -0.813669, 1.570796, 1.650339],accel_mss,speed_ms,0,blend_radius_m)
    speed_ms = 0.003
    movel([0.079543, -1.278628, -2.635558, -0.798202, 1.570796, 1.650339],accel_mss,speed_ms,0,blend_radius_m)
    speed_ms = 0.007
    movel([0.079179, -1.278689, -2.635524, -0.798176, 1.570796, 1.649975],accel_mss,speed_ms,0,blend_radius_m)
    movel([0.078923, -1.278520, -2.635620, -0.798249, 1.570796, 1.649719],accel_mss,speed_ms,0,blend_radius_m)
    movel([0.078964, -1.278213, -2.635794, -0.798382, 1.570796, 1.649760],accel_mss,speed_ms,0,blend_radius_m)
    movel([0.079062, -1.277767, -2.636048, -0.798574, 1.570796, 1.649858],accel_mss,speed_ms,0,blend_radius_m)
    movel([0.079237, -1.277126, -2.636411, -0.798852, 1.570796, 1.650033],accel_mss,speed_ms,0,blend_radius_m)
    movel([0.079964, -1.274485, -2.637904, -0.800000, 1.570796, 1.650760],accel_mss,speed_ms,0,blend_radius_m)
    movel([0.080502, -1.272286, -2.639140, -0.800963, 1.570796, 1.651299],accel_mss,speed_ms,0,blend_radius_m)
    movel([0.080891, -1.270390, -2.640202, -0.801798, 1.570796, 1.651687],accel_mss,speed_ms,0,blend_radius_m)
    movel([0.081149, -1.268687, -2.641151, -0.802551, 1.570796, 1.651945],accel_mss,speed_ms,0,blend_radius_m)
    movel([0.081193, -1.268418, -2.641300, -0.802671, 1.570796, 1.651989],accel_mss,speed_ms,0,blend_radius_m)
    movel([0.081325, -1.267944, -2.641564, -0.802881, 1.570796, 1.652121],accel_mss,speed_ms,0,blend_radius_m)
    movel([0.081671, -1.267648, -2.641728, -0.803013, 1.570796, 1.652467],accel_mss,speed_ms,0,blend_radius_m)
    movel([0.082725, -1.267358, -2.641889, -0.803142, 1.570796, 1.653521],accel_mss,speed_ms,0,blend_radius_m)
    movel([0.083753, -1.267116, -2.642023, -0.803250, 1.570796, 1.654549],accel_mss,speed_ms,0,blend_radius_m)
    movel([0.084117, -1.267131, -2.642015, -0.803243, 1.570796, 1.654913],accel_mss,speed_ms,0,blend_radius_m)
    movel([0.084231, -1.267507, -2.641806, -0.803076, 1.570796, 1.655027],accel_mss,speed_ms,0,blend_radius_m)
    movel([0.084115, -1.268003, -2.641531, -0.802855, 1.570796, 1.654911],accel_mss,speed_ms,0,blend_radius_m)
    movel([0.083731, -1.269313, -2.640802, -0.802274, 1.570796, 1.654527],accel_mss,speed_ms,0,blend_radius_m)
    movel([0.082917, -1.271780, -2.639424, -0.801185, 1.570796, 1.653713],accel_mss,speed_ms,0,blend_radius_m)
    movel([0.081808, -1.274705, -2.637780, -0.799904, 1.570796, 1.652604],accel_mss,speed_ms,0,blend_radius_m)
    movel([0.080667, -1.277499, -2.636200, -0.798690, 1.570796, 1.651463],accel_mss,speed_ms,0,blend_radius_m)
    movel([0.080149, -1.278313, -2.635737, -0.798338, 1.570796, 1.650946],accel_mss,speed_ms,0,blend_radius_m)
    movel([0.079543, -1.278628, -2.635558, -0.798202, 1.570796, 1.650339],accel_mss,speed_ms,0,blend_radius_m)
    speed_ms = 0.003
    movel([0.079543, -1.282169, -2.637215, -0.793005, 1.570796, 1.650339],accel_mss,speed_ms,0,blend_radius_m)
    speed_ms = 0.007
    movel([0.079179, -1.282229, -2.637180, -0.792979, 1.570796, 1.649975],accel_mss,speed_ms,0,blend_radius_m)
    movel([0.078923, -1.282061, -2.637277, -0.793051, 1.570796, 1.649719],accel_mss,speed_ms,0,blend_radius_m)
    movel([0.078964, -1.281755, -2.637452, -0.793183, 1.570796, 1.649760],accel_mss,speed_ms,0,blend_radius_m)
    movel([0.079062, -1.281309, -2.637706, -0.793374, 1.570796, 1.649858],accel_mss,speed_ms,0,blend_radius_m)
    movel([0.079237, -1.280670, -2.638071, -0.793649, 1.570796, 1.650033],accel_mss,speed_ms,0,blend_radius_m)
    movel([0.079964, -1.278035, -2.639568, -0.794787, 1.570796, 1.650760],accel_mss,speed_ms,0,blend_radius_m)
    movel([0.080502, -1.275839, -2.640808, -0.795741, 1.570796, 1.651299],accel_mss,speed_ms,0,blend_radius_m)
    movel([0.080891, -1.273947, -2.641872, -0.796569, 1.570796, 1.651687],accel_mss,speed_ms,0,blend_radius_m)
    movel([0.081149, -1.272248, -2.642824, -0.797317, 1.570796, 1.651945],accel_mss,speed_ms,0,blend_radius_m)
    movel([0.081193, -1.271980, -2.642974, -0.797435, 1.570796, 1.651989],accel_mss,speed_ms,0,blend_radius_m)
    movel([0.081325, -1.271506, -2.643239, -0.797644, 1.570796, 1.652121],accel_mss,speed_ms,0,blend_radius_m)
    movel([0.081671, -1.271211, -2.643403, -0.797774, 1.570796, 1.652467],accel_mss,speed_ms,0,blend_radius_m)
    movel([0.082725, -1.270922, -2.643565, -0.797902, 1.570796, 1.653521],accel_mss,speed_ms,0,blend_radius_m)
    movel([0.083753, -1.270680, -2.643700, -0.798009, 1.570796, 1.654549],accel_mss,speed_ms,0,blend_radius_m)
    movel([0.084117, -1.270696, -2.643691, -0.798002, 1.570796, 1.654913],accel_mss,speed_ms,0,blend_radius_m)
    movel([0.084231, -1.271070, -2.643482, -0.797836, 1.570796, 1.655027],accel_mss,speed_ms,0,blend_radius_m)
    movel([0.084115, -1.271565, -2.643206, -0.797618, 1.570796, 1.654911],accel_mss,speed_ms,0,blend_radius_m)
    movel([0.083731, -1.272872, -2.642475, -0.797042, 1.570796, 1.654527],accel_mss,speed_ms,0,blend_radius_m)
    movel([0.082917, -1.275335, -2.641092, -0.795962, 1.570796, 1.653713],accel_mss,speed_ms,0,blend_radius_m)
    movel([0.081808, -1.278254, -2.639443, -0.794692, 1.570796, 1.652604],accel_mss,speed_ms,0,blend_radius_m)
    movel([0.080667, -1.281042, -2.637859, -0.793489, 1.570796, 1.651463],accel_mss,speed_ms,0,blend_radius_m)
    movel([0.080149, -1.281855, -2.637395, -0.793140, 1.570796, 1.650946],accel_mss,speed_ms,0,blend_radius_m)
    movel([0.079543, -1.282169, -2.637215, -0.793005, 1.570796, 1.650339],accel_mss,speed_ms,0,blend_radius_m)
    speed_ms = 0.003
    movel([0.079543, -1.268182, -2.630539, -0.813669, 1.570796, 1.650339],accel_mss,speed_ms,0,blend_radius_m)
    speed_ms = 1.000
    movel([0.079543, -1.241590, -2.616802, -0.853997, 1.570796, 1.650339],accel_mss,speed_ms,0,blend_radius_m)
    movel([0.082583, -1.229496, -2.623251, -0.859642, 1.570796, 1.653379],accel_mss,speed_ms,0,blend_radius_m)
    movel([0.082583, -1.256233, -2.637147, -0.819009, 1.570796, 1.653379],accel_mss,speed_ms,0,blend_radius_m)
    speed_ms = 0.003
    movel([0.082583, -1.266747, -2.642228, -0.803414, 1.570796, 1.653379],accel_mss,speed_ms,0,blend_radius_m)
    speed_ms = 0.007
    movel([0.081950, -1.266899, -2.642143, -0.803347, 1.570796, 1.652747],accel_mss,speed_ms,0,blend_radius_m)
    movel([0.081416, -1.267011, -2.642081, -0.803297, 1.570796, 1.652213],accel_mss,speed_ms,0,blend_radius_m)
    movel([0.080713, -1.266884, -2.642152, -0.803353, 1.570796, 1.651509],accel_mss,speed_ms,0,blend_radius_m)
    movel([0.080445, -1.266352, -2.642446, -0.803590, 1.570796, 1.651241],accel_mss,speed_ms,0,blend_radius_m)
    movel([0.080325, -1.265372, -2.642988, -0.804029, 1.570796, 1.651122],accel_mss,speed_ms,0,blend_radius_m)
    movel([0.080346, -1.263733, -2.643892, -0.804764, 1.570796, 1.651143],accel_mss,speed_ms,0,blend_radius_m)
    movel([0.080457, -1.262170, -2.644750, -0.805468, 1.570796, 1.651254],accel_mss,speed_ms,0,blend_radius_m)
    movel([0.080748, -1.261614, -2.645055, -0.805720, 1.570796, 1.651544],accel_mss,speed_ms,0,blend_radius_m)
    movel([0.081360, -1.261197, -2.645283, -0.805908, 1.570796, 1.652157],accel_mss,speed_ms,0,blend_radius_m)
    movel([0.083606, -1.260361, -2.645741, -0.806288, 1.570796, 1.654402],accel_mss,speed_ms,0,blend_radius_m)
    movel([0.084619, -1.260004, -2.645935, -0.806450, 1.570796, 1.655415],accel_mss,speed_ms,0,blend_radius_m)
    movel([0.085490, -1.259712, -2.646095, -0.806582, 1.570796, 1.656286],accel_mss,speed_ms,0,blend_radius_m)
    movel([0.086238, -1.259471, -2.646226, -0.806692, 1.570796, 1.657035],accel_mss,speed_ms,0,blend_radius_m)
    movel([0.086357, -1.259687, -2.646108, -0.806594, 1.570796, 1.657153],accel_mss,speed_ms,0,blend_radius_m)
    movel([0.086285, -1.260113, -2.645876, -0.806400, 1.570796, 1.657081],accel_mss,speed_ms,0,blend_radius_m)
    movel([0.086211, -1.260416, -2.645711, -0.806263, 1.570796, 1.657007],accel_mss,speed_ms,0,blend_radius_m)
    movel([0.086111, -1.260869, -2.645463, -0.806057, 1.570796, 1.656908],accel_mss,speed_ms,0,blend_radius_m)
    movel([0.086001, -1.261377, -2.645185, -0.805827, 1.570796, 1.656797],accel_mss,speed_ms,0,blend_radius_m)
    movel([0.085898, -1.261868, -2.644916, -0.805605, 1.570796, 1.656694],accel_mss,speed_ms,0,blend_radius_m)
    movel([0.085795, -1.262410, -2.644619, -0.805360, 1.570796, 1.656592],accel_mss,speed_ms,0,blend_radius_m)
    movel([0.085689, -1.263075, -2.644254, -0.805060, 1.570796, 1.656486],accel_mss,speed_ms,0,blend_radius_m)
    movel([0.085596, -1.263754, -2.643880, -0.804755, 1.570796, 1.656393],accel_mss,speed_ms,0,blend_radius_m)
    movel([0.085529, -1.264334, -2.643561, -0.804494, 1.570796, 1.656326],accel_mss,speed_ms,0,blend_radius_m)
    movel([0.085380, -1.265451, -2.642945, -0.803993, 1.570796, 1.656176],accel_mss,speed_ms,0,blend_radius_m)
    movel([0.085137, -1.265878, -2.642709, -0.803802, 1.570796, 1.655933],accel_mss,speed_ms,0,blend_radius_m)
    movel([0.084672, -1.266164, -2.642551, -0.803675, 1.570796, 1.655468],accel_mss,speed_ms,0,blend_radius_m)
    movel([0.083253, -1.266575, -2.642323, -0.803491, 1.570796, 1.654049],accel_mss,speed_ms,0,blend_radius_m)
    movel([0.082583, -1.266747, -2.642228, -0.803414, 1.570796, 1.653379],accel_mss,speed_ms,0,blend_radius_m)
    speed_ms = 0.003
    movel([0.082583, -1.270312, -2.643905, -0.798172, 1.570796, 1.653379],accel_mss,speed_ms,0,blend_radius_m)
    speed_ms = 0.007
    movel([0.081950, -1.270464, -2.643820, -0.798105, 1.570796, 1.652747],accel_mss,speed_ms,0,blend_radius_m)
    movel([0.081416, -1.270576, -2.643758, -0.798055, 1.570796, 1.652213],accel_mss,speed_ms,0,blend_radius_m)
    movel([0.080713, -1.270449, -2.643829, -0.798112, 1.570796, 1.651509],accel_mss,speed_ms,0,blend_radius_m)
    movel([0.080445, -1.269918, -2.644124, -0.798347, 1.570796, 1.651241],accel_mss,speed_ms,0,blend_radius_m)
    movel([0.080325, -1.268940, -2.644668, -0.798781, 1.570796, 1.651122],accel_mss,speed_ms,0,blend_radius_m)
    movel([0.080346, -1.267304, -2.645574, -0.799511, 1.570796, 1.651143],accel_mss,speed_ms,0,blend_radius_m)
    movel([0.080457, -1.265745, -2.646435, -0.800209, 1.570796, 1.651254],accel_mss,speed_ms,0,blend_radius_m)
    movel([0.080748, -1.265190, -2.646741, -0.800459, 1.570796, 1.651544],accel_mss,speed_ms,0,blend_radius_m)
    movel([0.081360, -1.264773, -2.646970, -0.800646, 1.570796, 1.652157],accel_mss,speed_ms,0,blend_radius_m)
    movel([0.083606, -1.263938, -2.647429, -0.801022, 1.570796, 1.654402],accel_mss,speed_ms,0,blend_radius_m)
    movel([0.084619, -1.263582, -2.647624, -0.801183, 1.570796, 1.655415],accel_mss,speed_ms,0,blend_radius_m)
    movel([0.085490, -1.263291, -2.647784, -0.801314, 1.570796, 1.656286],accel_mss,speed_ms,0,blend_radius_m)
    movel([0.086238, -1.263050, -2.647916, -0.801423, 1.570796, 1.657035],accel_mss,speed_ms,0,blend_radius_m)
    movel([0.086357, -1.263266, -2.647797, -0.801325, 1.570796, 1.657153],accel_mss,speed_ms,0,blend_radius_m)
    movel([0.086285, -1.263692, -2.647564, -0.801133, 1.570796, 1.657081],accel_mss,speed_ms,0,blend_radius_m)
    movel([0.086211, -1.263993, -2.647398, -0.800997, 1.570796, 1.657007],accel_mss,speed_ms,0,blend_radius_m)
    movel([0.086111, -1.264445, -2.647150, -0.800793, 1.570796, 1.656908],accel_mss,speed_ms,0,blend_radius_m)
    movel([0.086001, -1.264953, -2.646871, -0.800565, 1.570796, 1.656797],accel_mss,speed_ms,0,blend_radius_m)
    movel([0.085898, -1.265443, -2.646601, -0.800345, 1.570796, 1.656694],accel_mss,speed_ms,0,blend_radius_m)
    movel([0.085795, -1.265984, -2.646303, -0.800102, 1.570796, 1.656592],accel_mss,speed_ms,0,blend_radius_m)
    movel([0.085689, -1.266647, -2.645937, -0.799805, 1.570796, 1.656486],accel_mss,speed_ms,0,blend_radius_m)
    movel([0.085596, -1.267325, -2.645563, -0.799502, 1.570796, 1.656393],accel_mss,speed_ms,0,blend_radius_m)
    movel([0.085529, -1.267904, -2.645242, -0.799243, 1.570796, 1.656326],accel_mss,speed_ms,0,blend_radius_m)
    movel([0.085380, -1.269019, -2.644624, -0.798746, 1.570796, 1.656176],accel_mss,speed_ms,0,blend_radius_m)
    movel([0.085137, -1.269445, -2.644387, -0.798557, 1.570796, 1.655933],accel_mss,speed_ms,0,blend_radius_m)
    movel([0.084672, -1.269730, -2.644229, -0.798430, 1.570796, 1.655468],accel_mss,speed_ms,0,blend_radius_m)
    movel([0.083253, -1.270140, -2.644000, -0.798248, 1.570796, 1.654049],accel_mss,speed_ms,0,blend_radius_m)
    movel([0.082583, -1.270312, -2.643905, -0.798172, 1.570796, 1.653379],accel_mss,speed_ms,0,blend_radius_m)
    speed_ms = 0.003
    movel([0.082583, -1.256233, -2.637147, -0.819009, 1.570796, 1.653379],accel_mss,speed_ms,0,blend_radius_m)
    speed_ms = 1.000
    movel([0.082583, -1.229496, -2.623251, -0.859642, 1.570796, 1.653379],accel_mss,speed_ms,0,blend_radius_m)
    movel([0.092310, -1.229064, -2.623478, -0.859847, 1.570796, 1.663107],accel_mss,speed_ms,0,blend_radius_m)
    movel([0.092310, -1.255806, -2.637380, -0.819203, 1.570796, 1.663107],accel_mss,speed_ms,0,blend_radius_m)
    speed_ms = 0.003
    movel([0.092310, -1.266323, -2.642463, -0.803604, 1.570796, 1.663107],accel_mss,speed_ms,0,blend_radius_m)
    speed_ms = 0.007
    movel([0.093445, -1.265797, -2.642754, -0.803839, 1.570796, 1.664242],accel_mss,speed_ms,0,blend_radius_m)
    movel([0.094363, -1.265473, -2.642933, -0.803984, 1.570796, 1.665160],accel_mss,speed_ms,0,blend_radius_m)
    movel([0.094630, -1.265516, -2.642909, -0.803964, 1.570796, 1.665426],accel_mss,speed_ms,0,blend_radius_m)
    movel([0.094539, -1.265873, -2.642711, -0.803804, 1.570796, 1.665336],accel_mss,speed_ms,0,blend_radius_m)
    movel([0.094064, -1.266107, -2.642582, -0.803700, 1.570796, 1.664861],accel_mss,speed_ms,0,blend_radius_m)
    movel([0.093493, -1.266293, -2.642479, -0.803617, 1.570796, 1.664289],accel_mss,speed_ms,0,blend_radius_m)
    movel([0.092792, -1.266495, -2.642367, -0.803527, 1.570796, 1.663589],accel_mss,speed_ms,0,blend_radius_m)
    movel([0.092422, -1.266550, -2.642337, -0.803502, 1.570796, 1.663219],accel_mss,speed_ms,0,blend_radius_m)
    movel([0.092310, -1.266323, -2.642463, -0.803604, 1.570796, 1.663107],accel_mss,speed_ms,0,blend_radius_m)
    speed_ms = 0.003
    movel([0.092310, -1.269888, -2.644140, -0.798360, 1.570796, 1.663107],accel_mss,speed_ms,0,blend_radius_m)
    speed_ms = 0.007
    movel([0.093445, -1.269364, -2.644432, -0.798593, 1.570796, 1.664242],accel_mss,speed_ms,0,blend_radius_m)
    movel([0.094363, -1.269040, -2.644612, -0.798737, 1.570796, 1.665160],accel_mss,speed_ms,0,blend_radius_m)
    movel([0.094630, -1.269083, -2.644588, -0.798718, 1.570796, 1.665426],accel_mss,speed_ms,0,blend_radius_m)
    movel([0.094539, -1.269440, -2.644390, -0.798559, 1.570796, 1.665336],accel_mss,speed_ms,0,blend_radius_m)
    movel([0.094064, -1.269673, -2.644260, -0.798456, 1.570796, 1.664861],accel_mss,speed_ms,0,blend_radius_m)
    movel([0.093493, -1.269859, -2.644157, -0.798373, 1.570796, 1.664289],accel_mss,speed_ms,0,blend_radius_m)
    movel([0.092792, -1.270060, -2.644045, -0.798284, 1.570796, 1.663589],accel_mss,speed_ms,0,blend_radius_m)
    movel([0.092422, -1.270115, -2.644014, -0.798259, 1.570796, 1.663219],accel_mss,speed_ms,0,blend_radius_m)
    movel([0.092310, -1.269888, -2.644140, -0.798360, 1.570796, 1.663107],accel_mss,speed_ms,0,blend_radius_m)
    speed_ms = 0.003
    movel([0.092310, -1.255806, -2.637380, -0.819203, 1.570796, 1.663107],accel_mss,speed_ms,0,blend_radius_m)
    speed_ms = 1.000
    movel([0.092310, -1.229064, -2.623478, -0.859847, 1.570796, 1.663107],accel_mss,speed_ms,0,blend_radius_m)
    movel([0.099561, -1.230071, -2.622948, -0.859370, 1.570796, 1.670358],accel_mss,speed_ms,0,blend_radius_m)
    movel([0.099561, -1.256801, -2.636837, -0.818751, 1.570796, 1.670358],accel_mss,speed_ms,0,blend_radius_m)
    speed_ms = 0.003
    movel([0.099561, -1.267312, -2.641914, -0.803162, 1.570796, 1.670358],accel_mss,speed_ms,0,blend_radius_m)
    speed_ms = 0.007
    movel([0.099947, -1.267089, -2.642038, -0.803262, 1.570796, 1.670743],accel_mss,speed_ms,0,blend_radius_m)
    movel([0.100597, -1.266887, -2.642150, -0.803352, 1.570796, 1.671393],accel_mss,speed_ms,0,blend_radius_m)
    movel([0.101348, -1.266671, -2.642270, -0.803448, 1.570796, 1.672144],accel_mss,speed_ms,0,blend_radius_m)
    movel([0.101677, -1.266608, -2.642305, -0.803476, 1.570796, 1.672473],accel_mss,speed_ms,0,blend_radius_m)
    movel([0.101808, -1.266783, -2.642208, -0.803398, 1.570796, 1.672604],accel_mss,speed_ms,0,blend_radius_m)
    movel([0.101464, -1.267006, -2.642084, -0.803299, 1.570796, 1.672260],accel_mss,speed_ms,0,blend_radius_m)
    movel([0.101097, -1.267158, -2.642000, -0.803231, 1.570796, 1.671893],accel_mss,speed_ms,0,blend_radius_m)
    movel([0.100604, -1.267336, -2.641901, -0.803152, 1.570796, 1.671400],accel_mss,speed_ms,0,blend_radius_m)
    movel([0.099927, -1.267559, -2.641777, -0.803052, 1.570796, 1.670723],accel_mss,speed_ms,0,blend_radius_m)
    movel([0.099533, -1.267588, -2.641761, -0.803040, 1.570796, 1.670330],accel_mss,speed_ms,0,blend_radius_m)
    movel([0.099561, -1.267312, -2.641914, -0.803162, 1.570796, 1.670358],accel_mss,speed_ms,0,blend_radius_m)
    speed_ms = 0.003
    movel([0.099561, -1.270876, -2.643590, -0.797922, 1.570796, 1.670358],accel_mss,speed_ms,0,blend_radius_m)
    speed_ms = 0.007
    movel([0.099947, -1.270654, -2.643714, -0.798021, 1.570796, 1.670743],accel_mss,speed_ms,0,blend_radius_m)
    movel([0.100597, -1.270452, -2.643827, -0.798110, 1.570796, 1.671393],accel_mss,speed_ms,0,blend_radius_m)
    movel([0.101348, -1.270236, -2.643947, -0.798206, 1.570796, 1.672144],accel_mss,speed_ms,0,blend_radius_m)
    movel([0.101677, -1.270173, -2.643982, -0.798234, 1.570796, 1.672473],accel_mss,speed_ms,0,blend_radius_m)
    movel([0.101808, -1.270348, -2.643885, -0.798156, 1.570796, 1.672604],accel_mss,speed_ms,0,blend_radius_m)
    movel([0.101464, -1.270571, -2.643761, -0.798058, 1.570796, 1.672260],accel_mss,speed_ms,0,blend_radius_m)
    movel([0.101097, -1.270722, -2.643676, -0.797991, 1.570796, 1.671893],accel_mss,speed_ms,0,blend_radius_m)
    movel([0.100604, -1.270900, -2.643577, -0.797912, 1.570796, 1.671400],accel_mss,speed_ms,0,blend_radius_m)
    movel([0.099927, -1.271123, -2.643453, -0.797813, 1.570796, 1.670723],accel_mss,speed_ms,0,blend_radius_m)
    movel([0.099533, -1.271151, -2.643437, -0.797801, 1.570796, 1.670330],accel_mss,speed_ms,0,blend_radius_m)
    movel([0.099561, -1.270876, -2.643590, -0.797922, 1.570796, 1.670358],accel_mss,speed_ms,0,blend_radius_m)
    speed_ms = 0.003
    movel([0.099561, -1.256801, -2.636837, -0.818751, 1.570796, 1.670358],accel_mss,speed_ms,0,blend_radius_m)
    speed_ms = 1.000
    movel([0.099561, -1.230071, -2.622948, -0.859370, 1.570796, 1.670358],accel_mss,speed_ms,0,blend_radius_m)
    movel([0.099464, -1.229425, -2.623288, -0.859676, 1.570796, 1.670261],accel_mss,speed_ms,0,blend_radius_m)
    movel([0.099464, -1.256163, -2.637185, -0.819041, 1.570796, 1.670261],accel_mss,speed_ms,0,blend_radius_m)
    speed_ms = 0.003
    movel([0.099464, -1.266678, -2.642266, -0.803445, 1.570796, 1.670261],accel_mss,speed_ms,0,blend_radius_m)
    speed_ms = 0.007
    movel([0.099864, -1.266398, -2.642421, -0.803570, 1.570796, 1.670661],accel_mss,speed_ms,0,blend_radius_m)
    movel([0.100140, -1.265931, -2.642679, -0.803779, 1.570796, 1.670936],accel_mss,speed_ms,0,blend_radius_m)
    movel([0.100356, -1.265081, -2.643149, -0.804159, 1.570796, 1.671153],accel_mss,speed_ms,0,blend_radius_m)
    movel([0.100640, -1.263246, -2.644160, -0.804983, 1.570796, 1.671436],accel_mss,speed_ms,0,blend_radius_m)
    movel([0.100880, -1.261605, -2.645060, -0.805724, 1.570796, 1.671677],accel_mss,speed_ms,0,blend_radius_m)
    movel([0.101009, -1.260957, -2.645415, -0.806017, 1.570796, 1.671805],accel_mss,speed_ms,0,blend_radius_m)
    movel([0.101145, -1.260582, -2.645620, -0.806187, 1.570796, 1.671942],accel_mss,speed_ms,0,blend_radius_m)
    movel([0.101358, -1.260292, -2.645778, -0.806319, 1.570796, 1.672154],accel_mss,speed_ms,0,blend_radius_m)
    movel([0.101658, -1.260042, -2.645915, -0.806432, 1.570796, 1.672454],accel_mss,speed_ms,0,blend_radius_m)
    movel([0.102128, -1.259955, -2.645962, -0.806472, 1.570796, 1.672924],accel_mss,speed_ms,0,blend_radius_m)
    movel([0.102340, -1.260116, -2.645874, -0.806399, 1.570796, 1.673136],accel_mss,speed_ms,0,blend_radius_m)
    movel([0.102446, -1.260348, -2.645747, -0.806293, 1.570796, 1.673242],accel_mss,speed_ms,0,blend_radius_m)
    movel([0.102458, -1.260728, -2.645540, -0.806121, 1.570796, 1.673254],accel_mss,speed_ms,0,blend_radius_m)
    movel([0.102379, -1.261416, -2.645164, -0.805809, 1.570796, 1.673176],accel_mss,speed_ms,0,blend_radius_m)
    movel([0.102123, -1.263031, -2.644278, -0.805080, 1.570796, 1.672919],accel_mss,speed_ms,0,blend_radius_m)
    movel([0.101853, -1.264772, -2.643319, -0.804297, 1.570796, 1.672649],accel_mss,speed_ms,0,blend_radius_m)
    movel([0.101798, -1.265520, -2.642906, -0.803962, 1.570796, 1.672594],accel_mss,speed_ms,0,blend_radius_m)
    movel([0.101884, -1.265846, -2.642726, -0.803816, 1.570796, 1.672681],accel_mss,speed_ms,0,blend_radius_m)
    movel([0.102127, -1.265892, -2.642701, -0.803796, 1.570796, 1.672923],accel_mss,speed_ms,0,blend_radius_m)
    movel([0.102418, -1.265924, -2.642683, -0.803782, 1.570796, 1.673214],accel_mss,speed_ms,0,blend_radius_m)
    movel([0.102637, -1.266057, -2.642610, -0.803722, 1.570796, 1.673433],accel_mss,speed_ms,0,blend_radius_m)
    movel([0.102685, -1.266335, -2.642456, -0.803598, 1.570796, 1.673481],accel_mss,speed_ms,0,blend_radius_m)
    movel([0.102479, -1.266979, -2.642099, -0.803311, 1.570796, 1.673275],accel_mss,speed_ms,0,blend_radius_m)
    movel([0.102314, -1.267259, -2.641944, -0.803186, 1.570796, 1.673111],accel_mss,speed_ms,0,blend_radius_m)
    movel([0.101871, -1.267582, -2.641764, -0.803042, 1.570796, 1.672667],accel_mss,speed_ms,0,blend_radius_m)
    movel([0.101580, -1.267799, -2.641644, -0.802946, 1.570796, 1.672376],accel_mss,speed_ms,0,blend_radius_m)
    movel([0.101261, -1.268211, -2.641416, -0.802763, 1.570796, 1.672057],accel_mss,speed_ms,0,blend_radius_m)
    movel([0.100848, -1.268752, -2.641115, -0.802523, 1.570796, 1.671644],accel_mss,speed_ms,0,blend_radius_m)
    movel([0.100469, -1.268999, -2.640977, -0.802413, 1.570796, 1.671265],accel_mss,speed_ms,0,blend_radius_m)
    movel([0.100136, -1.268960, -2.640999, -0.802430, 1.570796, 1.670932],accel_mss,speed_ms,0,blend_radius_m)
    movel([0.099864, -1.268617, -2.641190, -0.802582, 1.570796, 1.670660],accel_mss,speed_ms,0,blend_radius_m)
    movel([0.099641, -1.268371, -2.641327, -0.802692, 1.570796, 1.670438],accel_mss,speed_ms,0,blend_radius_m)
    movel([0.099334, -1.268343, -2.641342, -0.802704, 1.570796, 1.670130],accel_mss,speed_ms,0,blend_radius_m)
    movel([0.098951, -1.268375, -2.641324, -0.802690, 1.570796, 1.669747],accel_mss,speed_ms,0,blend_radius_m)
    movel([0.098703, -1.268278, -2.641378, -0.802733, 1.570796, 1.669500],accel_mss,speed_ms,0,blend_radius_m)
    movel([0.098605, -1.268048, -2.641506, -0.802835, 1.570796, 1.669401],accel_mss,speed_ms,0,blend_radius_m)
    movel([0.098652, -1.267700, -2.641699, -0.802990, 1.570796, 1.669448],accel_mss,speed_ms,0,blend_radius_m)
